           #FB_STATE_MONITOR:
               REGION MONITOR
                   IF #DATA.CMD_MON = 1 THEN
                       IF ("CycleInterrupt_Flag" = TRUE)
                       THEN
                           "CycleInterrupt_Flag" := FALSE;
                           #done := FALSE;
                           #statCMDStateDone := #FB_STATE_MONITOR;
                           FILL_BLK(IN := 16#00,
                                    COUNT := 20,
                                    OUT => #statSendData[0]);

                           #statSendData[0] := 16#02;
                           #statSendData[1] := 'M';
                           #statSendData[2] := 'O';
                           #statSendData[3] := 'N';
                           #statSendData[4] := 16#0D;

                           #statSendTxLength := 5;

                           #statSendReq := TRUE;
                       END_IF;
                   ELSE
                       #statCMDCount := 0;
                       #statCMDState := #statCMDState + 1;
                   END_IF;
               END_REGION MONITOR

           #FB_STATE_FAULT_CLEAR:
               REGION FAULT_CLEAR
                   IF #DATA.CMD_CLR = 1 THEN
                       IF ("CycleInterrupt_Flag" = TRUE)
                       THEN
                           "CycleInterrupt_Flag" := FALSE;
                           #done := FALSE;
                           #statCMDStateDone := #FB_STATE_FAULT_CLEAR;
                           FILL_BLK(IN := 16#00,
                                    COUNT := 20,
                                    OUT => #statSendData[0]);

                           #statSendData[0] := 16#02;
                           #statSendData[1] := 'C';
                           #statSendData[2] := 'L';
                           #statSendData[3] := 'R';
                           #statSendData[4] := 16#0D;

                           #statSendTxLength := 5;

                           #statSendReq := TRUE;
                       END_IF;
                       ELSE
                           #statCMDCount := 0;
                           #statCMDState := #statCMDState + 1;
                       END_IF;

               END_REGION FAULT_CLEAR

           #FB_STATE_REPORT_FAULT:
               REGION REPORT_FAULT
                   IF #DATA.CMD_FLT = 1 THEN
                       IF ("CycleInterrupt_Flag" = TRUE)
                       THEN
                           "CycleInterrupt_Flag" := FALSE;
                           #done := FALSE;
                           #statCMDStateDone := #FB_STATE_REPORT_FAULT;
                           FILL_BLK(IN := 16#00,
                                    COUNT := 20,
                                    OUT => #statSendData[0]);

                           #statSendData[0] := 16#02;
                           #statSendData[1] := 'F';
                           #statSendData[2] := 'L';
                           #statSendData[3] := 'T';
                           #statSendData[4] := 16#0D;

                           #statSendTxLength := 5;

                           #statSendReq := TRUE;
                       END_IF;
                   ELSE
                       #statCMDCount := 0;
                       #statCMDState := #statCMDState + 1;
                   END_IF;
               END_REGION REPORT_FAULT

           #FB_STATE_HV_STATUS:
               REGION HV_STATUS
                   IF #DATA.CMD_STAT = 1 THEN
                       IF ("CycleInterrupt_Flag" = TRUE)
                       THEN
                           "CycleInterrupt_Flag" := FALSE;
                           #done := FALSE;
                           #statCMDStateDone := #FB_STATE_HV_STATUS;
                           FILL_BLK(IN := 16#00,
                                    COUNT := 20,
                                    OUT => #statSendData[0]);

                           #statSendData[0] := 16#02;
                           #statSendData[1] := 'S';
                           #statSendData[2] := 'T';
                           #statSendData[3] := 'A';
                           #statSendData[4] := 'T';

                           #statSendData[5] := 16#0D;

                           #statSendTxLength := 6;

                           #statSendReq := TRUE;
                       END_IF;
                       ELSE
                           #statCMDCount := 0;
                           #statCMDState := #statCMDState + 1;
                       END_IF;
               END_REGION HV_STATUS

           #FB_STATE_X_RAY_ENABLE:
               REGION X_RAY_ENABLE
                   IF #DATA.CMD_ENBL = 1 THEN
                       IF ("CycleInterrupt_Flag" = TRUE)
                       THEN
                           "CycleInterrupt_Flag" := FALSE;
                           #done := FALSE;
                           #statCMDStateDone := #FB_STATE_WD_ENABLE;
                           FILL_BLK(IN := 16#00,
                                    COUNT := 20,
                                    OUT => #statSendData[0]);

                           #statSendData[0] := 16#02;
                           #statSendData[1] := 'E';
                           #statSendData[2] := 'N';
                           #statSendData[3] := 'B';
                           #statSendData[4] := 'L';

                           IF (#DATA.X_RAY_Enable = TRUE) THEN
                               #statSendData[5] := '1';
                           ELSE
                               #statSendData[5] := '0';
                           END_IF;
                           #statSendData[6] := 16#0D;
                           #statSendTxLength := 7;

                           #statSendReq := TRUE;
                       END_IF;
                   ELSE
                       #statCMDCount := 0;
                       #statCMDState := #statCMDState + 1;
                   END_IF;
               END_REGION X_RAY_ENABLE

           #FB_STATE_WD_TIMER:
               REGION WD_TIMER
                   IF #DATA.CMD_WDTE = 1 THEN
                       IF ("CycleInterrupt_Flag" = TRUE)
                       THEN
                           "CycleInterrupt_Flag" := FALSE;
                           #done := FALSE;
                           #statCMDStateDone := #FB_STATE_WD_TIMER;
                           FILL_BLK(IN := 16#00,
                                    COUNT := 20,
                                    OUT => #statSendData[0]);

                           #statSendData[0] := 16#02;
                           #statSendData[1] := 'W';
                           #statSendData[2] := 'D';
                           #statSendData[3] := 'T';
                           #statSendData[4] := 'E';
                           #statSendData[5] := 16#0D;
                           #statSendTxLength := 6;

                           #statSendReq := TRUE;
                       END_IF;
                   ELSE
                       #statCMDCount := 0;
                       #statCMDState := #statCMDState + 1;
                   END_IF;
               END_REGION WD_TIMER            

           #FB_STATE_COMM_PORT_ECHO:
               REGION PORT_ECHO
                   IF #DATA.CMD_FREV = 1 THEN
                       IF ("CycleInterrupt_Flag" = TRUE)
                       THEN
                           "CycleInterrupt_Flag" := FALSE;
                           #done := FALSE;
                           #statCMDStateDone := #FB_STATE_COMM_PORT_ECHO;
                              FILL_BLK(IN := 16#00,
                                       COUNT := 20,
                                       OUT => #statSendData[0]);

                           #statSendData[0] := 16#02;
                           #statSendData[1] := 'F';
                           #statSendData[2] := 'R';
                           #statSendData[3] := 'E';
                           #statSendData[4] := 'V';
                           #statSendData[5] := 16#0D;

                           #statSendTxLength := 6;
                           #statSendReq := TRUE;
                       END_IF;
                   ELSE
                       #statCMDCount := 0;
                       #statCMDState := #statCMDState + 1;
                   END_IF;
               END_REGION PORT_ECHO 

           #FB_STATE_WD_ENABLE:
               REGION WD_ENABLE
                   IF #DATA.CMD_WDOG = 1 THEN
                       IF ("CycleInterrupt_Flag" = TRUE)
                       THEN
                           "CycleInterrupt_Flag" := FALSE;
                           #done := FALSE;
                           #statCMDStateDone := #FB_STATE_WD_ENABLE;
                           FILL_BLK(IN := 16#00,
                                    COUNT := 20,
                                    OUT => #statSendData[0]);

                           #statSendData[0] := 16#02;
                           #statSendData[1] := 'W';
                           #statSendData[2] := 'D';
                           #statSendData[3] := 'O';
                           #statSendData[4] := 'G';

                           IF (#DATA.WDOG = TRUE) THEN
                               #statSendData[5] := '1';
                           ELSE
                               #statSendData[5] := '0';
                           END_IF;
                           #statSendData[6] := 16#0D;
                           #statSendTxLength := 7;

                           #statSendReq := TRUE;
                       END_IF;
                   ELSE
                       #statCMDCount := 0;
                       #statCMDState := #statCMDState + 1;
                   END_IF;
               END_REGION WD_ENABLE 

           #FB_STATE_WD_STATUS:
               REGION WD_STATUS
                   IF #DATA.CMD_WSTAT = 1 THEN
                       REGION Send WD_STATUS Request
                           IF ("CycleInterrupt_Flag" = TRUE)
                           THEN
                               #done := FALSE;
                               "CycleInterrupt_Flag" := FALSE;
                               #statCMDStateDone := #FB_STATE_WD_STATUS;
                               #done := FALSE;
                               FILL_BLK(IN := 16#00,
                               COUNT := 20,
                               OUT => #statSendData[0]);

                               FILL_BLK(IN := 16#00,
                                   COUNT := 50,
                                   OUT => #statRcvData[0]);
                                  #instReceiveP2P.LENGTH := 0;

                               #statSendData[0] := 16#02;
                               #statSendData[1] := 'W';
                               #statSendData[2] := 'S';
                               #statSendData[3] := 'T';
                               #statSendData[4] := 'A';
                               #statSendData[5] := 'T';

                               #statSendData[6] := 16#0D;

                               #statSendTxLength := 7;

                               #statSendReq := TRUE;
                           END_IF;
                       END_REGION Send WD_STATUS Request     
                   ELSE
                       #statCMDCount := 0;
                       #statCMDState := #FB_STATE_VOLTAGE_PROGRAMM;
                   END_IF;
               END_REGION WD_STATUS

           ELSE
               #statCMDState := #FB_STATE_VOLTAGE_PROGRAMM;

       END_CASE;


       IF #debug THEN
           // Statement section IF
           #statCMDCount := 0;
       END_IF;

    END_REGION STATE_MACHINE 

   REGION CALL COMMUNICATION INSTRUCTIONS

       "Send_P2P_DB"(REQ := #statSendReq,
                     "PORT" := #port,
                     BUFFER := #statSendData,
                     LENGTH := #statSendTxLength,
                     DONE => #statRS232TxDone,
                     ERROR => #statRS232Error,
                     STATUS => #statRS232Status);

       "Receive_P2P_DB"("PORT" := #port,
                        BUFFER := #statRcvData,
                        NDR => #statRS232Ndr,
                        ERROR => #statRS232Error,
                        STATUS => #statRS232Status,
                        LENGTH => #statSendRxLength);


   END_REGION CALL COMMUNICATION INSTRUCTIONS

   //Reset request has been sent
   IF #statRS232TxDone
   THEN
       #statSendReq := false;
   END_IF;

   IF #statRS232Ndr
   THEN
       #statStatus:= #statRS232Status;

       #statCMDCount := #statCMDCount + 1;

       IF (#statRS232Status = #STATUS_msg_timeout) OR (#statRS232Status = "STATUS_msg_CHAR_timeout") THEN
           CASE #statCMDState OF

               #FB_STATE_VOLTAGE_PROGRAMM:
                   REGION Recive Voltage Programm

                       IF #statSendRxLength = 8
                           AND #statRcvData[0] = #statSendData[0]
                           AND #statRcvData[1] = #statSendData[1]
                           AND #statRcvData[2] = #statSendData[2]
                           AND #statRcvData[3] = #statSendData[3]
                           AND #statRcvData[4] = #statSendData[4]
                           AND #statRcvData[5] = #statSendData[5]
                           AND #statRcvData[6] = #statSendData[6]
                           AND #statRcvData[7] = #statSendData[7]
                       THEN
                           #statCMDState := #statCMDState + 1;

                     //      IF NOT #DATA.CMD_CYCLE THEN
                           #DATA.CMD_VP := FALSE;
                           #DATA.CMD_VP_Ok := TRUE;
                      //     END_IF;
                       END_IF;
                   END_REGION Recive Voltage Programm       

               #FB_STATE_CURRENT_PROGRAMM:
                   REGION Recive Current Programm Request

                       IF #statSendRxLength = 8
                           AND #statRcvData[0] = #statSendData[0]
                           AND #statRcvData[1] = #statSendData[1]
                           AND #statRcvData[2] = #statSendData[2]
                           AND #statRcvData[3] = #statSendData[3]
                           AND #statRcvData[4] = #statSendData[4]
                           AND #statRcvData[5] = #statSendData[5]
                           AND #statRcvData[6] = #statSendData[6]
                       THEN
                           #statCMDState := #statCMDState + 1;
                   //        IF NOT #DATA.CMD_CYCLE THEN
                           #DATA.CMD_CP := FALSE;
                           #DATA.CMD_CP_Ok := TRUE;
                    //       END_IF;
                       END_IF;
                   END_REGION Recive Current Programm Request           

               #FB_STATE_MONITOR:
                   REGION Recive MONITOR Request
                       IF NOT #DATA.CMD_CYCLE THEN
                           #DATA.CMD_MON := FALSE;
                       END_IF;
                       IF #statSendRxLength = 21
                       THEN
                           //Вставить код для обработки ответа
                           //Преобразование V monitor
                           Chars_TO_Strg(Chars := #statRcvData,
          pChars := 1,
          Cnt := 4,
          Strg => #statString);
                           STRG_VAL(IN := #statString,
          FORMAT := 0,
          P := 1,
          OUT => #temp_Uint);
   #DATA.VP_Monitor := UINT_TO_REAL(#temp_Uint);
                           #DATA.VP_Monitor := #DATA.VP_Monitor / 10.0;

                           //Преобразование I monitor
                           Chars_TO_Strg(Chars := #statRcvData,
          pChars := 6,
          Cnt := 5,
          Strg => #statString);
                           STRG_VAL(IN := #statString,
          FORMAT := 0,
          P := 1,
          OUT => #temp_Uint);
                               #DATA.CP_Monitor := #temp_Uint;


                           //Преобразование T monitor
                           Chars_TO_Strg(Chars := #statRcvData,
          pChars := 12,
          Cnt := 4,
          Strg => #statString);
                           STRG_VAL(IN := #statString,
          FORMAT := 0,
          P := 1,
          OUT => #temp_Uint);
                           #DATA.T_Monitor := UINT_TO_REAL(#temp_Uint);
                           #DATA.T_Monitor := #DATA.T_Monitor / 10.0;

                           //Преобразование Filament monitor
                           Chars_TO_Strg(Chars := #statRcvData,
          pChars := 17,
          Cnt := 4,
          Strg => #statString);
                           STRG_VAL(IN := #statString,
          FORMAT := 0,
          P := 1,
          OUT => #temp_Uint);
                           #DATA.FIL_Monitor := #temp_Uint;

                           #statCMDState := #statCMDState + 1;
                       END_IF;
                   END_REGION Recive MONITOR Request 

               #FB_STATE_FAULT_CLEAR:
                   REGION Recive FAULT_CLEAR Request
                       IF NOT #DATA.CMD_CYCLE THEN
                           #DATA.CMD_CLR := FALSE;
                       END_IF;
                       IF #statRcvData[0] = #statSendData[0]
                           AND #statRcvData[1] = #statSendData[1]
                           AND #statRcvData[2] = #statSendData[2]
                           AND #statRcvData[3] = #statSendData[3]
                           AND #statRcvData[4] = #statSendData[4]
                       THEN
                           #statCMDCount := 0;
                           #statCMDState := #statCMDState + 1;
                       END_IF;
                   END_REGION Recive FAULT_CLEAR Request   

               #FB_STATE_REPORT_FAULT:
                   REGION Recive REPORT_FAULT Request
                       IF NOT #DATA.CMD_CYCLE THEN
                           #DATA.CMD_FLT := FALSE;
                       END_IF;
                       IF #statSendRxLength = 19
                       THEN
                           //Вставить код для обработки ответа
                           IF #statRcvData[1] = '1' THEN
                               #DATA.FLT[0] := TRUE;
                           ELSE
                               #DATA.FLT[0] := FALSE;
                           END_IF;

                           IF #statRcvData[3] = '1' THEN
                               #DATA.FLT[1] := TRUE;
                           ELSE
                               #DATA.FLT[1] := FALSE;
                           END_IF;

                           IF #statRcvData[5] = '1' THEN
                               #DATA.FLT[2] := TRUE;
                           ELSE
                               #DATA.FLT[2] := FALSE;
                           END_IF;

                           IF #statRcvData[7] = '1' THEN
                               #DATA.FLT[3] := TRUE;
                           ELSE
                               #DATA.FLT[3] := FALSE;
                           END_IF;

                           IF #statRcvData[9] = '1' THEN
                               #DATA.FLT[4] := TRUE;
                           ELSE
                               #DATA.FLT[4] := FALSE;
                           END_IF;

                           IF #statRcvData[11] = '1' THEN
                               #DATA.FLT[5] := TRUE;
                           ELSE
                               #DATA.FLT[5] := FALSE;
                           END_IF;

                           IF #statRcvData[13] = '1' THEN
                               #DATA.FLT[6] := TRUE;
                           ELSE
                               #DATA.FLT[6] := FALSE;
                           END_IF;

                           IF #statRcvData[15] = '1' THEN
                               #DATA.FLT[7] := TRUE;
                           ELSE
                               #DATA.FLT[7] := FALSE;
                           END_IF;

                           IF #statRcvData[17] = '1' THEN
                               #DATA.FLT[8] := TRUE;
                           ELSE
                               #DATA.FLT[8] := FALSE;
                           END_IF;

                           #statCMDState := #statCMDState + 1;
                       END_IF;
                   END_REGION Recive REPORT_FAULT Request   

               #FB_STATE_HV_STATUS:
                   REGION Recive MONITOR Reques                
                       IF NOT #DATA.CMD_CYCLE THEN
                           #DATA.CMD_STAT := FALSE;
                       END_IF;
                       IF #statSendRxLength = 3
                       THEN
                           IF (#statRcvData[1] = '1') THEN
                               #DATA.X_RAY_Status := TRUE;
                           ELSE
                               #DATA.X_RAY_Status := FALSE;
                           END_IF;
                           #statCMDCount := 0;
                           #statCMDState := #statCMDState + 1;
                       END_IF;
                   END_REGION Recive HV_STATUS Request  

               #FB_STATE_X_RAY_ENABLE:
                   REGION Recive X_RAY_ENABLE Request
                       IF NOT #DATA.CMD_CYCLE THEN
                           #DATA.CMD_ENBL := FALSE;
                       END_IF;
                       IF  (#statSendRxLength = 7)
                           AND #statRcvData[1] = #statSendData[1]
                           AND #statRcvData[2] = #statSendData[2]
                           AND #statRcvData[3] = #statSendData[3]
                           AND #statRcvData[4] = #statSendData[4]
                       THEN
                           IF #statRcvData[5] = '1' THEN
                               #DATA.X_RAY_Enable := TRUE;
                           ELSE
                               #DATA.X_RAY_Enable := FALSE;
                           END_IF;
                           #statCMDCount := 0;
                           #statCMDState := #statCMDState + 1;
                       END_IF;
                   END_REGION Recive X_RAY_ENABLE Request 

               #FB_STATE_WD_TIMER:
                   REGION Recive WD_TIMER Request
                       IF NOT #DATA.CMD_CYCLE THEN
                           #DATA.CMD_WDTE := FALSE;
                       END_IF;
                       IF (#statSendRxLength = 4)
                           AND #statRcvData[1] = 'O'
                           AND #statRcvData[2] = 'K'
                       THEN
                           #DATA.WDTE := TRUE;
                           #statCMDCount := 0;
                           #statCMDState := #statCMDState + 1;
                       END_IF;
                   END_REGION Recive WD_TIMER Request 

               #FB_STATE_COMM_PORT_ECHO:
                   REGION Recive PORT_ECHO Request
                       IF NOT #DATA.CMD_CYCLE THEN
                           #DATA.CMD_FREV := FALSE;
                       END_IF;
                       IF #statSendRxLength = 6
                           AND #statRcvData[1] = 16#32
                           AND #statRcvData[2] = 16#30
                           AND #statRcvData[3] = 16#30
                           AND #statRcvData[4] = 16#30
                       THEN
                           //Вставить код для обработки ответа
                           #DATA.FREV := TRUE;
                           #statCMDCount := 0;
                           #statCMDState := #statCMDState + 1;
                       END_IF;
                   END_REGION Recive PORT_ECHO Request  

               #FB_STATE_WD_ENABLE:
                   REGION Recive WD_ENABLE Request
                       IF NOT #DATA.CMD_CYCLE THEN
                           #DATA.CMD_WDOG := FALSE;
                       END_IF;
                       IF #statSendRxLength = 7
                           AND #statRcvData[0] = #statSendData[0]
                           AND #statRcvData[1] = #statSendData[1]
                           AND #statRcvData[2] = #statSendData[2]
                           AND #statRcvData[3] = #statSendData[3]
                           AND #statRcvData[4] = #statSendData[4]
                       THEN
                           IF #statRcvData[5] = '1' THEN
                               #DATA.WDOG := TRUE;
                           ELSE
                               #DATA.WDOG := FALSE;
                           END_IF;
                           #statCMDCount := 0;
                           #statCMDState := #statCMDState + 1;
                       END_IF;
                       END_REGION Recive WD_ENABLE Request  

               #FB_STATE_WD_STATUS:
                   REGION Recive WD_STATUS    
                       IF #statSendRxLength = 3
                       THEN
                           IF NOT #DATA.CMD_CYCLE THEN
                               #DATA.CMD_WSTAT := FALSE;
                           END_IF;
                           IF (#statRcvData[1] = '1') THEN
                               #DATA.WDOG_Status := TRUE;
                           ELSE
                               #DATA.WDOG_Status := FALSE;
                           END_IF;
                           #statCMDState := #FB_STATE_VOLTAGE_PROGRAMM;
                       END_IF;
                   END_REGION Recive WD_STATUS
               ELSE
                   REGION undefined state        
                       #statCMDState := #FB_STATE_VOLTAGE_PROGRAMM;
                   END_REGION undefined state    
           END_CASE;
           #statCMDCount := 0;
           #statError := FALSE;
       ELSE
           #statError := TRUE;
           #statCMDCount := #statCMDCount +1;
           IF #statCMDCount >= "CountERR" THEN
               #statCMDState := #FB_STATE_NO_PROCESSING;
               #DATA.DiagnosticCMD[#statCMDState].status := #statStatus;
               #DATA.DiagnosticCMD[#statCMDState].count := #statCMDCount;
           END_IF;
       END_IF;
   END_IF;

   REGION OUTPUT  
       REGION Write static values to outputs

           #error := #statError;
           #status := #statStatus;
           IF (NOT #error)
               AND ((#statRS232TxDone AND #debug) OR (#statRS232Ndr AND (#statStatus <> #ERR_Response_Generator)))
           THEN
               #done := TRUE;
           END_IF;

           #DATA.DiagnosticCMD[#statCMDState].status := #status;
           #DATA.DiagnosticCMD[#statCMDState].count := #statCMDCount + 1;

           #done_CMD := #statCMDState;

           ENO := TRUE;

       END_REGION Write static values to outputs
   END_REGION OUTPUTS
END_FUNCTION_BLOCK

FUNCTION_BLOCK "GenOperate"   // FB8, LAD
{ S7_Optimized_Access := 'TRUE' }
VERSION : 0.1
   VAR_INPUT
      cmdXRAY : Bool;
      interLock : Bool;
      statusGEN : Bool;
      resset : Bool;
      HW_PORT : Port;
      SelGen1 : Bool;
      SelGen2 : Bool;
   END_VAR
   VAR_OUTPUT
      "X-RAY_HL" : Bool;
      POWER_Status : Bool;
      Fault : Bool;
      Ready : Bool;
      Status : Word;
   END_VAR
   VAR_IN_OUT
      DATA_Generator : "typeGeneratorDATA";
   END_VAR
   VAR
      err_CMD_Generator : Bool;
      status_CMD_Gnerator : UInt;
      err_Check_Presset : Bool;
      done_CMD_Generator : Bool;
      status_POWER_OK : Bool;
      status_Delta_VP : Real;
      status_Delta_CP : Real;
      reset_Generator : Bool;
      noACK : Bool;
      Front1 : Bool;
      Front2 : Bool;
      Rise1 : Bool;
   END_VAR
   VAR_TEMP   // added for the SCL form of the ladder/FBD networks
      _w1 : Bool;
      _w2 : Bool;
      _w3 : Bool;
   END_VAR
BEGIN

REGION Network 1: Command HV Status
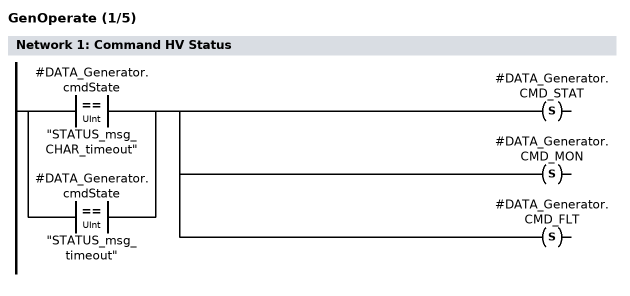
   RUNG wire#powerrail
      { S7_Templates := "SrcType := UInt" } EQ_Contact(in1 := #DATA_Generator.cmdState, in2 := "STATUS_msg_CHAR_timeout")
      wire#w1
      S_Coil( #DATA_Generator.CMD_STAT )
   END_RUNG
   RUNG wire#powerrail
      { S7_Templates := "SrcType := UInt" } EQ_Contact(in1 := #DATA_Generator.cmdState, in2 := "STATUS_msg_timeout")
   END_RUNG wire#w1
   RUNG wire#w1
      S_Coil( #DATA_Generator.CMD_MON )
   END_RUNG
   RUNG wire#w1
      S_Coil( #DATA_Generator.CMD_FLT )
   END_RUNG
   // the same network as SCL:
   IF (#DATA_Generator.cmdState = "STATUS_msg_CHAR_timeout") OR (#DATA_Generator.cmdState = "STATUS_msg_timeout") THEN
       #DATA_Generator.CMD_STAT := TRUE;
       #DATA_Generator.CMD_MON := TRUE;
       #DATA_Generator.CMD_FLT := TRUE;
   END_IF;
END_REGION

REGION Network 2: Когда нет ответа от генератора, то сбрасываем блок работы с генератором
   // Проверка соединения с генератором. Если при выполнении команды получаем ошибку по таймауту ответа от генератора, то сбрасываем интерфейс обмена с генератором, включаем режим DEBUG (при отутствии ответа от генератора не останавливаем обмен), цстанавливаем циклический обмен и запускаем команду на получения ECHO. Как только по команде получения ECHO мы получаем ответ от генератора, то сбрасываем команду на получения ECHO, а выставляем команду Monitor и WD. Получаем фактическое значение напряжения и тока генератора, читаем сторожевой таймер
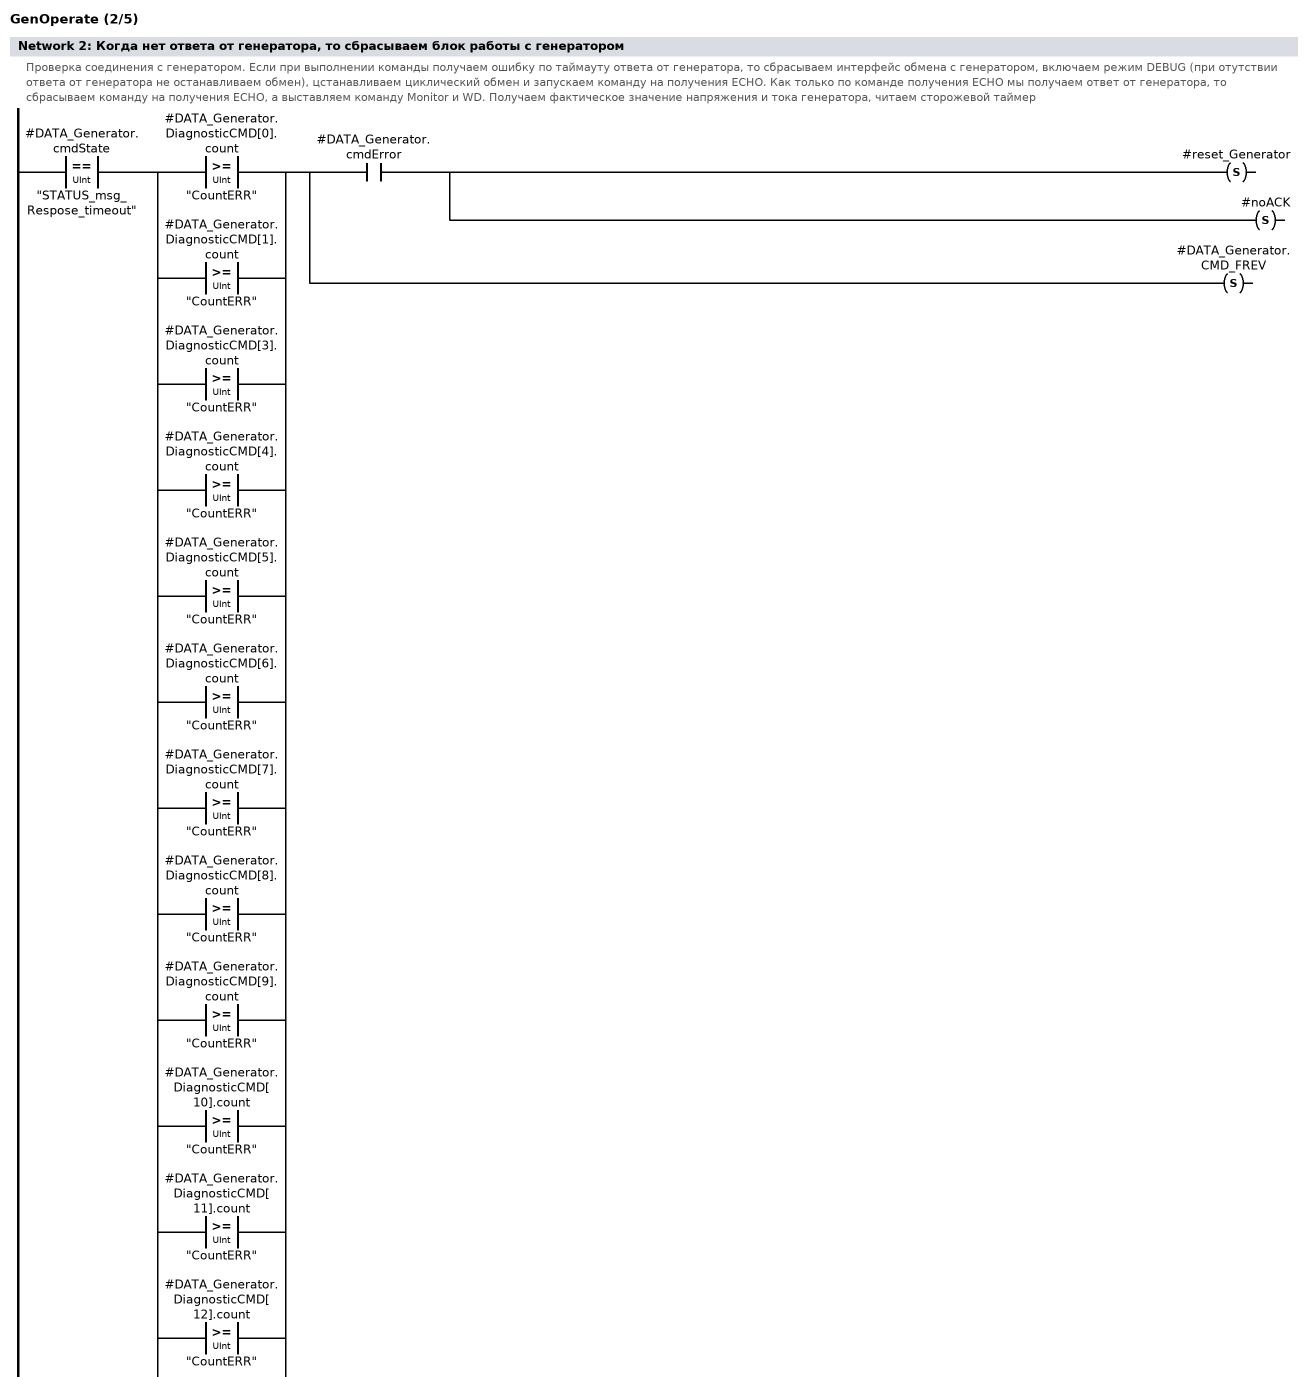
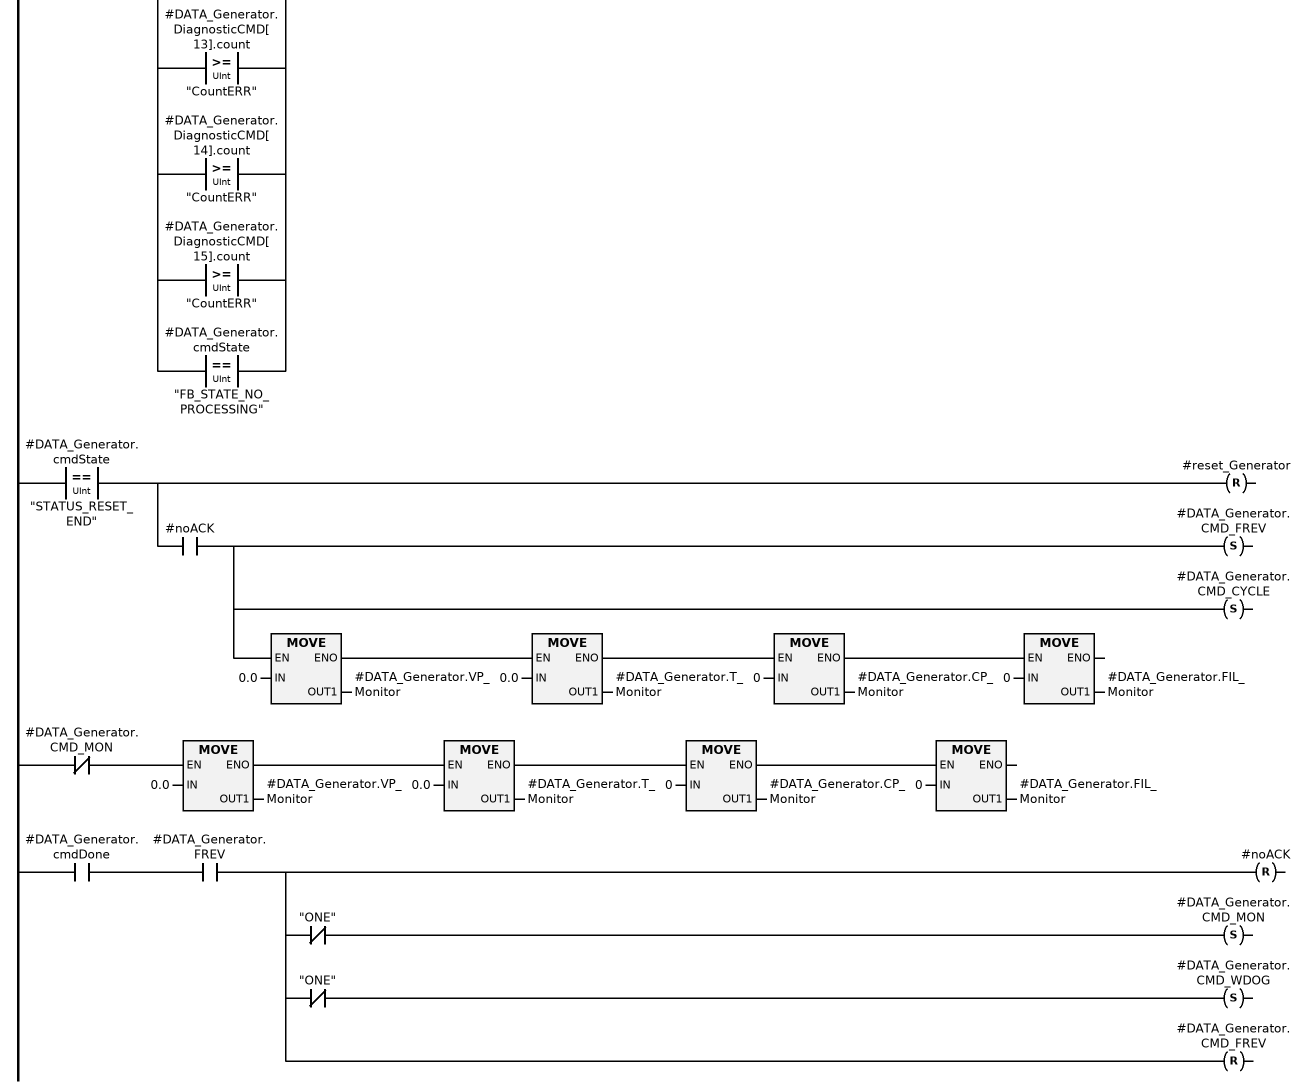
   RUNG wire#powerrail
      { S7_Templates := "SrcType := UInt" } EQ_Contact(in1 := #DATA_Generator.cmdState, in2 := "STATUS_msg_Respose_timeout")
      wire#w1
      { S7_Templates := "SrcType := UInt" } GE_Contact(in1 := #DATA_Generator.DiagnosticCMD[0].count, in2 := "CountERR")
      wire#w2
      Contact( #DATA_Generator.cmdError )
      wire#w3
      S_Coil( #reset_Generator )
   END_RUNG
   RUNG wire#w1
      { S7_Templates := "SrcType := UInt" } GE_Contact(in1 := #DATA_Generator.DiagnosticCMD[1].count, in2 := "CountERR")
   END_RUNG wire#w2
   RUNG wire#w1
      { S7_Templates := "SrcType := UInt" } GE_Contact(in1 := #DATA_Generator.DiagnosticCMD[3].count, in2 := "CountERR")
   END_RUNG wire#w2
   RUNG wire#w1
      { S7_Templates := "SrcType := UInt" } GE_Contact(in1 := #DATA_Generator.DiagnosticCMD[4].count, in2 := "CountERR")
   END_RUNG wire#w2
   RUNG wire#w1
      { S7_Templates := "SrcType := UInt" } GE_Contact(in1 := #DATA_Generator.DiagnosticCMD[5].count, in2 := "CountERR")
   END_RUNG wire#w2
   RUNG wire#w1
      { S7_Templates := "SrcType := UInt" } GE_Contact(in1 := #DATA_Generator.DiagnosticCMD[6].count, in2 := "CountERR")
   END_RUNG wire#w2
   RUNG wire#w1
      { S7_Templates := "SrcType := UInt" } GE_Contact(in1 := #DATA_Generator.DiagnosticCMD[7].count, in2 := "CountERR")
   END_RUNG wire#w2
   RUNG wire#w1
      { S7_Templates := "SrcType := UInt" } GE_Contact(in1 := #DATA_Generator.DiagnosticCMD[8].count, in2 := "CountERR")
   END_RUNG wire#w2
   RUNG wire#w1
      { S7_Templates := "SrcType := UInt" } GE_Contact(in1 := #DATA_Generator.DiagnosticCMD[9].count, in2 := "CountERR")
   END_RUNG wire#w2
   RUNG wire#w1
      { S7_Templates := "SrcType := UInt" } GE_Contact(in1 := #DATA_Generator.DiagnosticCMD[10].count, in2 := "CountERR")
   END_RUNG wire#w2
   RUNG wire#w1
      { S7_Templates := "SrcType := UInt" } GE_Contact(in1 := #DATA_Generator.DiagnosticCMD[11].count, in2 := "CountERR")
   END_RUNG wire#w2
   RUNG wire#w1
      { S7_Templates := "SrcType := UInt" } GE_Contact(in1 := #DATA_Generator.DiagnosticCMD[12].count, in2 := "CountERR")
   END_RUNG wire#w2
   RUNG wire#w1
      { S7_Templates := "SrcType := UInt" } GE_Contact(in1 := #DATA_Generator.DiagnosticCMD[13].count, in2 := "CountERR")
   END_RUNG wire#w2
   RUNG wire#w1
      { S7_Templates := "SrcType := UInt" } GE_Contact(in1 := #DATA_Generator.DiagnosticCMD[14].count, in2 := "CountERR")
   END_RUNG wire#w2
   RUNG wire#w1
      { S7_Templates := "SrcType := UInt" } GE_Contact(in1 := #DATA_Generator.DiagnosticCMD[15].count, in2 := "CountERR")
   END_RUNG wire#w2
   RUNG wire#w1
      { S7_Templates := "SrcType := UInt" } EQ_Contact(in1 := #DATA_Generator.cmdState, in2 := "FB_STATE_NO_PROCESSING")
   END_RUNG wire#w2
   RUNG wire#w3
      S_Coil( #noACK )
   END_RUNG
   RUNG wire#w2
      S_Coil( #DATA_Generator.CMD_FREV )
   END_RUNG
   RUNG wire#powerrail
      { S7_Templates := "SrcType := UInt" } EQ_Contact(in1 := #DATA_Generator.cmdState, in2 := "STATUS_RESET_END")
      wire#w4
      R_Coil( #reset_Generator )
   END_RUNG
   RUNG wire#w4
      Contact( #noACK )
      wire#w5
      S_Coil( #DATA_Generator.CMD_FREV )
   END_RUNG
   RUNG wire#w5
      S_Coil( #DATA_Generator.CMD_CYCLE )
   END_RUNG
   RUNG wire#w5
      Move(in := 0.0, out1 => #DATA_Generator.VP_Monitor)
      Move(in := 0.0, out1 => #DATA_Generator.T_Monitor)
      Move(in := 0, out1 => #DATA_Generator.CP_Monitor)
      Move(in := 0, out1 => #DATA_Generator.FIL_Monitor)
   END_RUNG
   RUNG wire#powerrail
      I_Contact( #DATA_Generator.CMD_MON )
      Move(in := 0.0, out1 => #DATA_Generator.VP_Monitor)
      Move(in := 0.0, out1 => #DATA_Generator.T_Monitor)
      Move(in := 0, out1 => #DATA_Generator.CP_Monitor)
      Move(in := 0, out1 => #DATA_Generator.FIL_Monitor)
   END_RUNG
   RUNG wire#powerrail
      Contact( #DATA_Generator.cmdDone )
      Contact( #DATA_Generator.FREV )
      wire#w6
      R_Coil( #noACK )
   END_RUNG
   RUNG wire#w6
      I_Contact( "ONE" )
      S_Coil( #DATA_Generator.CMD_MON )
   END_RUNG
   RUNG wire#w6
      I_Contact( "ONE" )
      S_Coil( #DATA_Generator.CMD_WDOG )
   END_RUNG
   RUNG wire#w6
      R_Coil( #DATA_Generator.CMD_FREV )
   END_RUNG
   // the same network as SCL:
   #_w1 := (#DATA_Generator.cmdState = "STATUS_msg_Respose_timeout") AND ((#DATA_Generator.DiagnosticCMD[0].count >= "CountERR") OR (#DATA_Generator.DiagnosticCMD[1].count >= "CountERR") OR (#DATA_Generator.DiagnosticCMD[3].count >= "CountERR") OR (#DATA_Generator.DiagnosticCMD[4].count >= "CountERR") OR (#DATA_Generator.DiagnosticCMD[5].count >= "CountERR") OR (#DATA_Generator.DiagnosticCMD[6].count >= "CountERR") OR (#DATA_Generator.DiagnosticCMD[7].count >= "CountERR") OR (#DATA_Generator.DiagnosticCMD[8].count >= "CountERR") OR (#DATA_Generator.DiagnosticCMD[9].count >= "CountERR") OR (#DATA_Generator.DiagnosticCMD[10].count >= "CountERR") OR (#DATA_Generator.DiagnosticCMD[11].count >= "CountERR") OR (#DATA_Generator.DiagnosticCMD[12].count >= "CountERR") OR (#DATA_Generator.DiagnosticCMD[13].count >= "CountERR") OR (#DATA_Generator.DiagnosticCMD[14].count >= "CountERR") OR (#DATA_Generator.DiagnosticCMD[15].count >= "CountERR") OR (#DATA_Generator.cmdState = "FB_STATE_NO_PROCESSING"));
   IF #_w1 AND #DATA_Generator.cmdError THEN
       #reset_Generator := TRUE;
       #noACK := TRUE;
   END_IF;
   IF #_w1 THEN #DATA_Generator.CMD_FREV := TRUE; END_IF;
   #_w2 := #DATA_Generator.cmdState = "STATUS_RESET_END";
   IF #_w2 THEN #reset_Generator := FALSE; END_IF;
   IF #_w2 AND #noACK THEN
       #DATA_Generator.CMD_FREV := TRUE;
       #DATA_Generator.CMD_CYCLE := TRUE;
       #DATA_Generator.VP_Monitor := 0.0;
       #DATA_Generator.T_Monitor := 0.0;
       #DATA_Generator.CP_Monitor := 0;
       #DATA_Generator.FIL_Monitor := 0;
   END_IF;
   IF NOT #DATA_Generator.CMD_MON THEN
       #DATA_Generator.VP_Monitor := 0.0;
       #DATA_Generator.T_Monitor := 0.0;
       #DATA_Generator.CP_Monitor := 0;
       #DATA_Generator.FIL_Monitor := 0;
   END_IF;
   #_w3 := #DATA_Generator.cmdDone AND #DATA_Generator.FREV;
   IF #_w3 THEN #noACK := FALSE; END_IF;
   IF #_w3 AND NOT "ONE" THEN
       #DATA_Generator.CMD_MON := TRUE;
       #DATA_Generator.CMD_WDOG := TRUE;
   END_IF;
   IF #_w3 THEN #DATA_Generator.CMD_FREV := FALSE; END_IF;
END_REGION

REGION Network 3: Включение X-RAY
   // По сигналу устанавливаем:
   // 1. Команду программирования Напряжения и Тока в генераторе
   // 2. Сброс статуса выполнения команды на программирование Напряджения и Тока
   // 3. После выполнения команды программирования Напряжения и Тока выставляем статус выполнения команд
   // 4. Пос статусу выполнения команды устанавливаем команду на включение генаратора
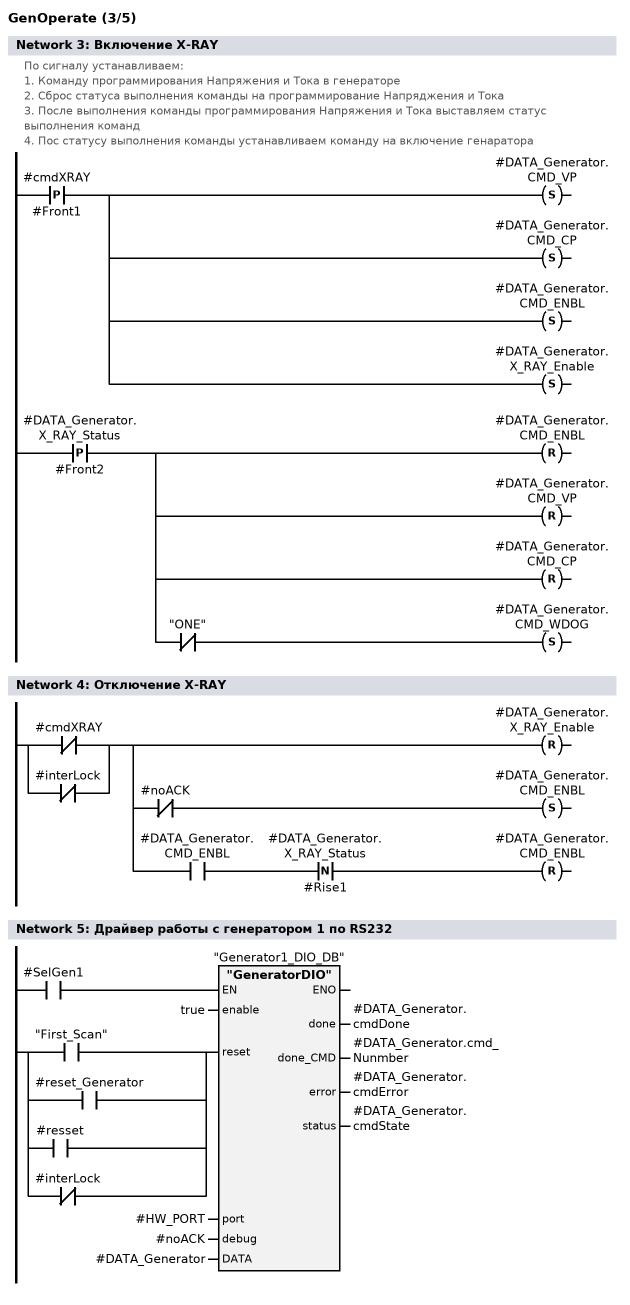
   RUNG wire#powerrail
      P_Contact(operand := #cmdXRAY, bit := #Front1)
      wire#w1
      S_Coil( #DATA_Generator.CMD_VP )
   END_RUNG
   RUNG wire#w1
      S_Coil( #DATA_Generator.CMD_CP )
   END_RUNG
   RUNG wire#w1
      S_Coil( #DATA_Generator.CMD_ENBL )
   END_RUNG
   RUNG wire#w1
      S_Coil( #DATA_Generator.X_RAY_Enable )
   END_RUNG
   RUNG wire#powerrail
      P_Contact(operand := #DATA_Generator.X_RAY_Status, bit := #Front2)
      wire#w2
      R_Coil( #DATA_Generator.CMD_ENBL )
   END_RUNG
   RUNG wire#w2
      R_Coil( #DATA_Generator.CMD_VP )
   END_RUNG
   RUNG wire#w2
      R_Coil( #DATA_Generator.CMD_CP )
   END_RUNG
   RUNG wire#w2
      I_Contact( "ONE" )
      S_Coil( #DATA_Generator.CMD_WDOG )
   END_RUNG
   // the same network as SCL:
   #_w1 := #cmdXRAY AND NOT #Front1;   // rising edge of #cmdXRAY
   #Front1 := #cmdXRAY;
   IF #_w1 THEN
       #DATA_Generator.CMD_VP := TRUE;
       #DATA_Generator.CMD_CP := TRUE;
       #DATA_Generator.CMD_ENBL := TRUE;
       #DATA_Generator.X_RAY_Enable := TRUE;
   END_IF;
   #_w2 := #DATA_Generator.X_RAY_Status AND NOT #Front2;   // rising edge of #DATA_Generator.X_RAY_Status
   #Front2 := #DATA_Generator.X_RAY_Status;
   IF #_w2 THEN
       #DATA_Generator.CMD_ENBL := FALSE;
       #DATA_Generator.CMD_VP := FALSE;
       #DATA_Generator.CMD_CP := FALSE;
   END_IF;
   IF #_w2 AND NOT "ONE" THEN #DATA_Generator.CMD_WDOG := TRUE; END_IF;
END_REGION

REGION Network 4: Отключение X-RAY
   RUNG wire#powerrail
      I_Contact( #cmdXRAY )
      wire#w1
      R_Coil( #DATA_Generator.X_RAY_Enable )
   END_RUNG
   RUNG wire#powerrail
      I_Contact( #interLock )
   END_RUNG wire#w1
   RUNG wire#w1
      I_Contact( #noACK )
      S_Coil( #DATA_Generator.CMD_ENBL )
   END_RUNG
   RUNG wire#w1
      Contact( #DATA_Generator.CMD_ENBL )
      N_Contact(operand := #DATA_Generator.X_RAY_Status, bit := #Rise1)
      R_Coil( #DATA_Generator.CMD_ENBL )
   END_RUNG
   // the same network as SCL:
   #_w1 := NOT #cmdXRAY OR NOT #interLock;
   IF #_w1 THEN #DATA_Generator.X_RAY_Enable := FALSE; END_IF;
   IF #_w1 AND NOT #noACK THEN #DATA_Generator.CMD_ENBL := TRUE; END_IF;
   #_w2 := #_w1 AND #DATA_Generator.CMD_ENBL AND NOT #DATA_Generator.X_RAY_Status AND #Rise1;   // falling edge of #DATA_Generator.X_RAY_Status
   #Rise1 := #DATA_Generator.X_RAY_Status;
   IF #_w2 THEN #DATA_Generator.CMD_ENBL := FALSE; END_IF;
END_REGION

REGION Network 5: Драйвер работы с генератором 1 по RS232
   RUNG wire#powerrail
      Contact( #SelGen1 )
      "Generator1_DIO_DB"(reset := wire#w1, enable := true, port := #HW_PORT, debug := #noACK, DATA := #DATA_Generator, done => #DATA_Generator.cmdDone, done_CMD => #DATA_Generator.cmd_Nunmber, error => #DATA_Generator.cmdError, status => #DATA_Generator.cmdState)
   END_RUNG
   RUNG wire#powerrail
      Contact( "First_Scan" )
   END_RUNG wire#w1
   RUNG wire#powerrail
      Contact( #reset_Generator )
   END_RUNG wire#w1
   RUNG wire#powerrail
      Contact( #resset )
   END_RUNG wire#w1
   RUNG wire#powerrail
      I_Contact( #interLock )
   END_RUNG wire#w1
   // the same network as SCL:
   IF #SelGen1 THEN
       "Generator1_DIO_DB"(enable := true,   // "GeneratorDIO"
                           reset := "First_Scan" OR #reset_Generator OR #resset OR NOT #interLock,
                           port := #HW_PORT,
                           debug := #noACK,
                           DATA := #DATA_Generator,
                           done => #DATA_Generator.cmdDone,
                           done_CMD => #DATA_Generator.cmd_Nunmber,
                           error => #DATA_Generator.cmdError,
                           status => #DATA_Generator.cmdState);
   END_IF;
END_REGION

REGION Network 6: Драйвер работы с генератором 2 по RS232
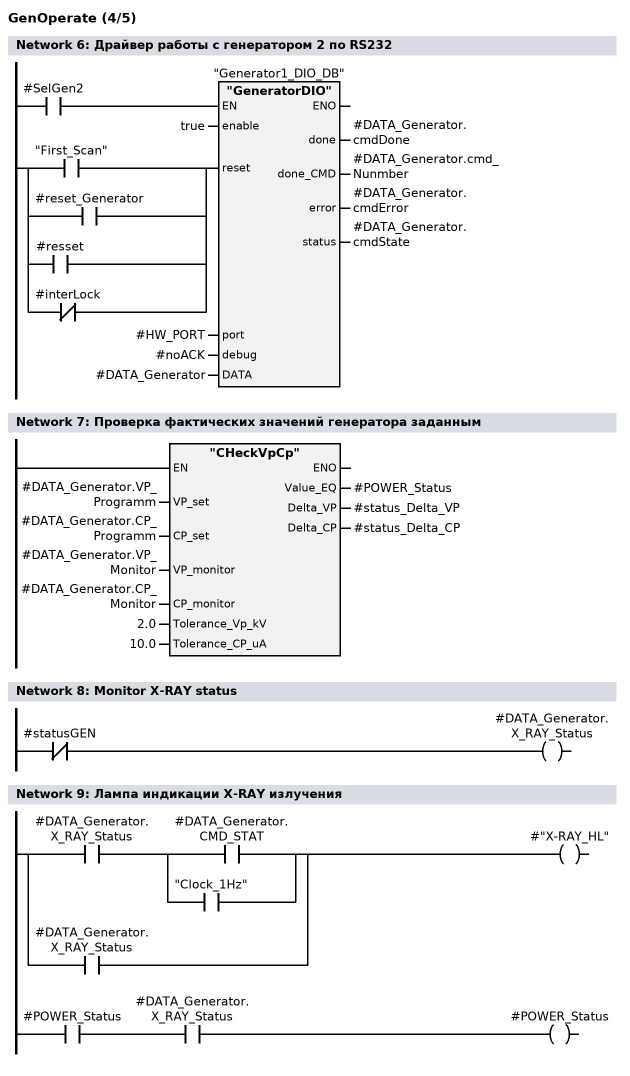
   RUNG wire#powerrail
      Contact( #SelGen2 )
      "Generator1_DIO_DB"(reset := wire#w1, enable := true, port := #HW_PORT, debug := #noACK, DATA := #DATA_Generator, done => #DATA_Generator.cmdDone, done_CMD => #DATA_Generator.cmd_Nunmber, error => #DATA_Generator.cmdError, status => #DATA_Generator.cmdState)
   END_RUNG
   RUNG wire#powerrail
      Contact( "First_Scan" )
   END_RUNG wire#w1
   RUNG wire#powerrail
      Contact( #reset_Generator )
   END_RUNG wire#w1
   RUNG wire#powerrail
      Contact( #resset )
   END_RUNG wire#w1
   RUNG wire#powerrail
      I_Contact( #interLock )
   END_RUNG wire#w1
   // the same network as SCL:
   IF #SelGen2 THEN
       "Generator1_DIO_DB"(enable := true,   // "GeneratorDIO"
                           reset := "First_Scan" OR #reset_Generator OR #resset OR NOT #interLock,
                           port := #HW_PORT,
                           debug := #noACK,
                           DATA := #DATA_Generator,
                           done => #DATA_Generator.cmdDone,
                           done_CMD => #DATA_Generator.cmd_Nunmber,
                           error => #DATA_Generator.cmdError,
                           status => #DATA_Generator.cmdState);
   END_IF;
END_REGION

REGION Network 7: Проверка фактических значений генератора заданным
   RUNG wire#powerrail
      "CHeckVpCp"(VP_set := #DATA_Generator.VP_Programm, CP_set := #DATA_Generator.CP_Programm, VP_monitor := #DATA_Generator.VP_Monitor, CP_monitor := #DATA_Generator.CP_Monitor, Tolerance_Vp_kV := 2.0, Tolerance_CP_uA := 10.0, Value_EQ => #POWER_Status, Delta_VP => #status_Delta_VP, Delta_CP => #status_Delta_CP)
   END_RUNG
   // the same network as SCL:
   "CHeckVpCp"(VP_set := #DATA_Generator.VP_Programm,
               CP_set := #DATA_Generator.CP_Programm,
               VP_monitor := #DATA_Generator.VP_Monitor,
               CP_monitor := #DATA_Generator.CP_Monitor,
               Tolerance_Vp_kV := 2.0,
               Tolerance_CP_uA := 10.0,
               Value_EQ => #POWER_Status,
               Delta_VP => #status_Delta_VP,
               Delta_CP => #status_Delta_CP);
END_REGION

REGION Network 8: Monitor X-RAY status
   RUNG wire#powerrail
      I_Contact( #statusGEN )
      Coil( #DATA_Generator.X_RAY_Status )
   END_RUNG
   // the same network as SCL:
   #DATA_Generator.X_RAY_Status := NOT #statusGEN;
END_REGION

REGION Network 9: Лампа индикации X-RAY излучения
   RUNG wire#powerrail
      Contact( #DATA_Generator.X_RAY_Status )
      wire#w1
      Contact( #DATA_Generator.CMD_STAT )
      wire#w2
      Coil( #"X-RAY_HL" )
   END_RUNG
   RUNG wire#w1
      Contact( "Clock_1Hz" )
   END_RUNG wire#w2
   RUNG wire#powerrail
      Contact( #DATA_Generator.X_RAY_Status )
   END_RUNG wire#w2
   RUNG wire#powerrail
      Contact( #POWER_Status )
      Contact( #DATA_Generator.X_RAY_Status )
      Coil( #POWER_Status )
   END_RUNG
   // the same network as SCL:
   #"X-RAY_HL" := (#DATA_Generator.X_RAY_Status AND (#DATA_Generator.CMD_STAT OR "Clock_1Hz")) OR #DATA_Generator.X_RAY_Status;
   #POWER_Status := #POWER_Status AND #DATA_Generator.X_RAY_Status;
END_REGION

REGION Network 10 (SCL): Проверка ошибок от генератора
   IF #DATA_Generator.FLT[0] = TRUE
       OR #DATA_Generator.FLT[1] = TRUE
       OR #DATA_Generator.FLT[2] = TRUE
       OR #DATA_Generator.FLT[3] = TRUE
       OR #DATA_Generator.FLT[4] = TRUE
       OR #DATA_Generator.FLT[5] = TRUE
       OR #DATA_Generator.FLT[6] = TRUE
       OR #DATA_Generator.FLT[7] = TRUE
       OR #DATA_Generator.FLT[8] = TRUE
       OR #DATA_Generator.FLT[8] = TRUE
       OR #DATA_Generator.cmdError = TRUE
   THEN
       #Fault := TRUE;
   ELSE
       #Fault := FALSE;
   END_IF;
END_REGION

REGION Network 11: Проверка готовности генератора
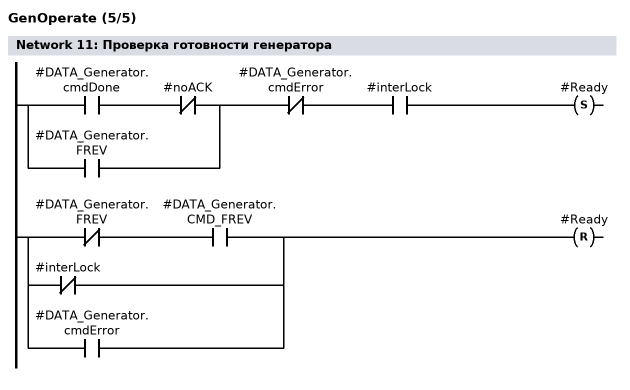
   RUNG wire#powerrail
      Contact( #DATA_Generator.cmdDone )
      I_Contact( #noACK )
      wire#w1
      I_Contact( #DATA_Generator.cmdError )
      Contact( #interLock )
      S_Coil( #Ready )
   END_RUNG
   RUNG wire#powerrail
      Contact( #DATA_Generator.FREV )
   END_RUNG wire#w1
   RUNG wire#powerrail
      I_Contact( #DATA_Generator.FREV )
      Contact( #DATA_Generator.CMD_FREV )
      wire#w2
      R_Coil( #Ready )
   END_RUNG
   RUNG wire#powerrail
      I_Contact( #interLock )
   END_RUNG wire#w2
   RUNG wire#powerrail
      Contact( #DATA_Generator.cmdError )
   END_RUNG wire#w2
   // the same network as SCL:
   IF ((#DATA_Generator.cmdDone AND NOT #noACK) OR #DATA_Generator.FREV) AND NOT #DATA_Generator.cmdError AND #interLock THEN
       #Ready := TRUE;
   END_IF;
   IF (NOT #DATA_Generator.FREV AND #DATA_Generator.CMD_FREV) OR NOT #interLock OR #DATA_Generator.cmdError THEN
       #Ready := FALSE;
   END_IF;
END_REGION

REGION Network 12 (SCL)
   #Status := #DATA_Generator.cmdState;
END_REGION
END_FUNCTION_BLOCK

FUNCTION "CheckPresset" : Void   // FC1, SCL
{ S7_Optimized_Access := 'TRUE' }
VERSION : 0.1
   VAR_INPUT
      VP_max_kV : Real;
      VP_min_kV : Real;
      CP_max_uA : UInt;
      CP_min_uA : UInt;
      "FEED_max_%" : UInt;
      "FEED_min_%" : UInt;
   END_VAR
   VAR_OUTPUT
      error : Bool;
   END_VAR
   VAR_IN_OUT
      DATA_MIDLE : "typePresset";
      DATA_LOW : "typePresset";
      DATA_HIGH : "typePresset";
   END_VAR
   VAR_TEMP
      error_check : Bool;
   END_VAR
BEGIN
   #error_check := TRUE;
   // Проверка диапазона напряжений МАКСИМУМ
   IF #DATA_LOW.VP > #VP_max_kV THEN
       // Statement section IF
       #DATA_LOW.VP := #VP_max_kV;
   ELSE
       #error_check := FALSE;
   END_IF;

   IF #DATA_MIDLE.VP > #VP_max_kV THEN
       // Statement section IF
       #DATA_MIDLE.VP := #VP_max_kV;
   ELSE
       #error_check := FALSE;
   END_IF;

   IF #DATA_HIGH.VP > #VP_max_kV THEN
       // Statement section IF
       #DATA_HIGH.VP := #VP_max_kV;
   ELSE
       #error_check := FALSE;
   END_IF;

   // Проверка диапазона напряжений МИНИМУМ
   IF #DATA_LOW.VP < #VP_min_kV THEN
       // Statement section IF
       #DATA_LOW.VP := #VP_min_kV;
   ELSE
       #error_check := FALSE;
   END_IF;

   IF #DATA_MIDLE.VP < #VP_min_kV THEN
       // Statement section IF
       #DATA_MIDLE.VP := #VP_min_kV;
   ELSE
       #error_check := FALSE;
   END_IF;

   IF #DATA_HIGH.VP < #VP_min_kV THEN
       // Statement section IF
       #DATA_HIGH.VP := #VP_min_kV;
   ELSE
       #error_check := FALSE;
   END_IF;

   // Проверка диапазона токов МАКСИМУМ
   IF #DATA_LOW.CP > #CP_max_uA THEN
       // Statement section IF
       #DATA_LOW.CP := #CP_max_uA;
   ELSE
       #error_check := FALSE;
   END_IF;

   IF #DATA_MIDLE.CP > #CP_max_uA THEN
       // Statement section IF
       #DATA_MIDLE.CP := #CP_max_uA;
   ELSE
       #error_check := FALSE;
   END_IF;

   IF #DATA_HIGH.CP > #CP_max_uA THEN
       // Statement section IF
       #DATA_HIGH.CP := #CP_max_uA;
   ELSE
       #error_check := FALSE;
   END_IF;

   // Проверка диапазона токов МИНИМУМ
   IF #DATA_LOW.CP < #CP_min_uA THEN
       // Statement section IF
       #DATA_LOW.CP := #CP_min_uA;
   ELSE
       #error_check := FALSE;
   END_IF;

   IF #DATA_MIDLE.CP < #CP_min_uA THEN
       // Statement section IF
       #DATA_MIDLE.CP := #CP_min_uA;
   ELSE
       #error_check := FALSE;
   END_IF;

   IF #DATA_HIGH.CP < #CP_min_uA THEN
       // Statement section IF
       #DATA_HIGH.CP := #CP_min_uA;
   ELSE
       #error_check := FALSE;
   END_IF;

   // Проверка диапазона скорости шторки МАКСИМУМ
   IF #DATA_LOW.Velocity > #"FEED_max_%" THEN
       // Statement section IF
       #DATA_LOW.Velocity := #"FEED_max_%";
   ELSE
       #error_check := FALSE;
   END_IF;


   IF #DATA_MIDLE.Velocity > #"FEED_max_%" THEN
       // Statement section IF
       #DATA_MIDLE.Velocity := #"FEED_max_%";
   ELSE
       #error_check := FALSE;
   END_IF;

   IF #DATA_HIGH.Velocity > #"FEED_max_%" THEN
       // Statement section IF
       #DATA_HIGH.Velocity := #"FEED_max_%";
   ELSE
       #error_check := FALSE;
   END_IF;

   // Проверка диапазона скорости шторки МИНИМУМ
   IF #DATA_LOW.Velocity < #"FEED_min_%" THEN
       // Statement section IF
       #DATA_LOW.Velocity := #"FEED_min_%";
   ELSE
       #error_check := FALSE;
   END_IF;


   IF #DATA_MIDLE.Velocity < #"FEED_min_%" THEN
       // Statement section IF
       #DATA_MIDLE.Velocity := #"FEED_min_%";
   ELSE
       #error_check := FALSE;
   END_IF;

   IF #DATA_HIGH.Velocity < #"FEED_min_%" THEN
       // Statement section IF
       #DATA_HIGH.Velocity := #"FEED_min_%";
   ELSE
       #error_check := FALSE;
   END_IF;

   #error := #error_check;
END_FUNCTION

FUNCTION "CHeckVpCp" : Void   // FC3, SCL
{ S7_Optimized_Access := 'TRUE' }
VERSION : 0.1
   VAR_INPUT
      VP_set : Real;
      CP_set : UInt;
      VP_monitor : Real;
      CP_monitor : Real;
      Tolerance_Vp_kV : Real;
      Tolerance_CP_uA : Real;
   END_VAR
   VAR_OUTPUT
      Value_EQ : Bool;
      Delta_VP : Real;
      Delta_CP : Real;
   END_VAR
   VAR_TEMP
      DeltaVP : Real;
      DeltaCP : Real;
   END_VAR
BEGIN
   #DeltaVP := ABS(#VP_set - #VP_monitor);
   #DeltaCP := ABS(#CP_set - #CP_monitor);

   IF #VP_set = 0.0 OR #CP_set = 0 THEN
       #Value_EQ := FALSE;
       RETURN;
   END_IF;

   IF (#DeltaVP < #Tolerance_Vp_kV) AND (#DeltaCP < #Tolerance_CP_uA) THEN
       // Statement section IF
       #Value_EQ:=TRUE;
   ELSE
       #Value_EQ := FALSE;
   END_IF;

   #Delta_VP := #DeltaVP;
   #Delta_CP := #DeltaCP;
END_FUNCTION

FUNCTION "LoadPresset" : Void   // FC4, SCL
{ S7_Optimized_Access := 'TRUE' }
VERSION : 0.1
   VAR_INPUT
      N_Presset : UInt;
      DATA_from : "typePresset";
   END_VAR
   VAR_OUTPUT
      DATA_to : "typeGeneratorDATA";
   END_VAR
BEGIN
   #DATA_to.VP_Programm := #DATA_from.VP;
   #DATA_to.CP_Programm := #DATA_from.CP;
END_FUNCTION

FUNCTION "GeneratorStage" : Void   // FC9, LAD
{ S7_Optimized_Access := 'TRUE' }
VERSION : 0.1
   VAR_IN_OUT
      DATA_Generator1 : "typeGeneratorDATA";
      DATA_Generator2 : "typeGeneratorDATA";
   END_VAR
   VAR_TEMP
      err_Check_Presset : Bool;
      HL_XRAY_1 : Bool;
      HL_XRAY_2 : Bool;
   END_VAR
BEGIN

REGION Network 1: Проверка уставок
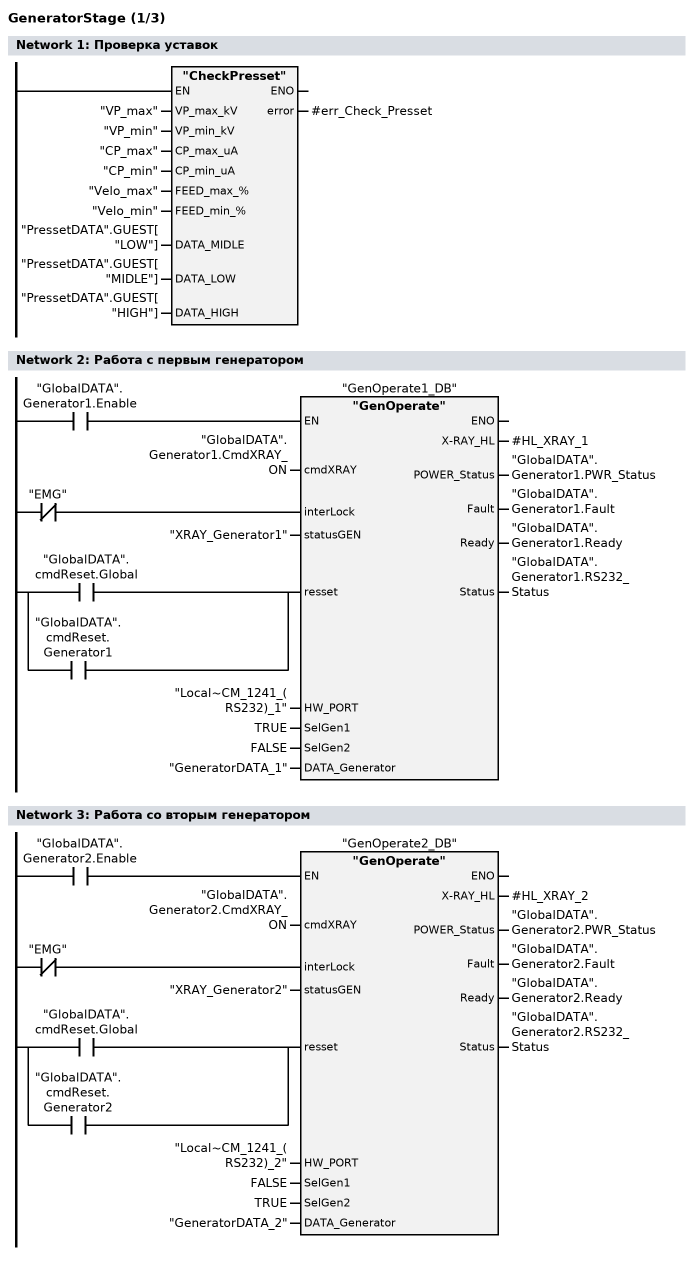
   RUNG wire#powerrail
      "CheckPresset"(VP_max_kV := "VP_max", VP_min_kV := "VP_min", CP_max_uA := "CP_max", CP_min_uA := "CP_min", "FEED_max_%" := "Velo_max", "FEED_min_%" := "Velo_min", DATA_MIDLE := "PressetDATA".GUEST["LOW"], DATA_LOW := "PressetDATA".GUEST["MIDLE"], DATA_HIGH := "PressetDATA".GUEST["HIGH"], error => #err_Check_Presset)
   END_RUNG
   // the same network as SCL:
   "CheckPresset"(VP_max_kV := "VP_max",
                  VP_min_kV := "VP_min",
                  CP_max_uA := "CP_max",
                  CP_min_uA := "CP_min",
                  "FEED_max_%" := "Velo_max",
                  "FEED_min_%" := "Velo_min",
                  DATA_MIDLE := "PressetDATA".GUEST["LOW"],
                  DATA_LOW := "PressetDATA".GUEST["MIDLE"],
                  DATA_HIGH := "PressetDATA".GUEST["HIGH"],
                  error => #err_Check_Presset);
END_REGION

REGION Network 2: Работа с первым генератором
   RUNG wire#powerrail
      Contact( "GlobalDATA".Generator1.Enable )
      "GenOperate1_DB"(interLock := wire#w1, resset := wire#w2, cmdXRAY := "GlobalDATA".Generator1.CmdXRAY_ON, statusGEN := "XRAY_Generator1", HW_PORT := "Local~CM_1241_(RS232)_1", SelGen1 := TRUE, SelGen2 := FALSE, DATA_Generator := "GeneratorDATA_1", "X-RAY_HL" => #HL_XRAY_1, POWER_Status => "GlobalDATA".Generator1.PWR_Status, Fault => "GlobalDATA".Generator1.Fault, Ready => "GlobalDATA".Generator1.Ready, Status => "GlobalDATA".Generator1.RS232_Status)
   END_RUNG
   RUNG wire#powerrail
      I_Contact( "EMG" )
   END_RUNG wire#w1
   RUNG wire#powerrail
      Contact( "GlobalDATA".cmdReset.Global )
   END_RUNG wire#w2
   RUNG wire#powerrail
      Contact( "GlobalDATA".cmdReset.Generator1 )
   END_RUNG wire#w2
   // the same network as SCL:
   IF "GlobalDATA".Generator1.Enable THEN
       "GenOperate1_DB"(cmdXRAY := "GlobalDATA".Generator1.CmdXRAY_ON,   // "GenOperate"
                        interLock := NOT "EMG",
                        statusGEN := "XRAY_Generator1",
                        resset := "GlobalDATA".cmdReset.Global OR "GlobalDATA".cmdReset.Generator1,
                        HW_PORT := "Local~CM_1241_(RS232)_1",
                        SelGen1 := TRUE,
                        SelGen2 := FALSE,
                        DATA_Generator := "GeneratorDATA_1",
                        "X-RAY_HL" => #HL_XRAY_1,
                        POWER_Status => "GlobalDATA".Generator1.PWR_Status,
                        Fault => "GlobalDATA".Generator1.Fault,
                        Ready => "GlobalDATA".Generator1.Ready,
                        Status => "GlobalDATA".Generator1.RS232_Status);
   END_IF;
END_REGION

REGION Network 3: Работа со вторым генератором
   RUNG wire#powerrail
      Contact( "GlobalDATA".Generator2.Enable )
      "GenOperate2_DB"(interLock := wire#w1, resset := wire#w2, cmdXRAY := "GlobalDATA".Generator2.CmdXRAY_ON, statusGEN := "XRAY_Generator2", HW_PORT := "Local~CM_1241_(RS232)_2", SelGen1 := FALSE, SelGen2 := TRUE, DATA_Generator := "GeneratorDATA_2", "X-RAY_HL" => #HL_XRAY_2, POWER_Status => "GlobalDATA".Generator2.PWR_Status, Fault => "GlobalDATA".Generator2.Fault, Ready => "GlobalDATA".Generator2.Ready, Status => "GlobalDATA".Generator2.RS232_Status)
   END_RUNG
   RUNG wire#powerrail
      I_Contact( "EMG" )
   END_RUNG wire#w1
   RUNG wire#powerrail
      Contact( "GlobalDATA".cmdReset.Global )
   END_RUNG wire#w2
   RUNG wire#powerrail
      Contact( "GlobalDATA".cmdReset.Generator2 )
   END_RUNG wire#w2
   // the same network as SCL:
   IF "GlobalDATA".Generator2.Enable THEN
       "GenOperate2_DB"(cmdXRAY := "GlobalDATA".Generator2.CmdXRAY_ON,   // "GenOperate"
                        interLock := NOT "EMG",
                        statusGEN := "XRAY_Generator2",
                        resset := "GlobalDATA".cmdReset.Global OR "GlobalDATA".cmdReset.Generator2,
                        HW_PORT := "Local~CM_1241_(RS232)_2",
                        SelGen1 := FALSE,
                        SelGen2 := TRUE,
                        DATA_Generator := "GeneratorDATA_2",
                        "X-RAY_HL" => #HL_XRAY_2,
                        POWER_Status => "GlobalDATA".Generator2.PWR_Status,
                        Fault => "GlobalDATA".Generator2.Fault,
                        Ready => "GlobalDATA".Generator2.Ready,
                        Status => "GlobalDATA".Generator2.RS232_Status);
   END_IF;
END_REGION

REGION Network 4 (SCL): Передача в глобальный блок данных состояния генератора 1
   "GlobalDATA".Generator1.CP_monitor := #DATA_Generator1.CP_Monitor;
   "GlobalDATA".Generator1.VP_monitor := #DATA_Generator1.VP_Monitor;
   "GlobalDATA".Generator1.T_monitor := #DATA_Generator1.T_Monitor;
   "GlobalDATA".Generator1.CP := #DATA_Generator1.CP_Programm;
   "GlobalDATA".Generator1.VP := #DATA_Generator1.VP_Programm;
   "GlobalDATA".Generator1.XRAY_Status := #DATA_Generator1.X_RAY_Status;
   "GlobalDATA".Generator1.FLT[0] := #DATA_Generator1.FLT[0];
   "GlobalDATA".Generator1.FLT[1] := #DATA_Generator1.FLT[1];
   "GlobalDATA".Generator1.FLT[2] := #DATA_Generator1.FLT[2];
   "GlobalDATA".Generator1.FLT[3] := #DATA_Generator1.FLT[3];
   "GlobalDATA".Generator1.FLT[4] := #DATA_Generator1.FLT[4];
   "GlobalDATA".Generator1.FLT[5] := #DATA_Generator1.FLT[5];
   "GlobalDATA".Generator1.FLT[6] := #DATA_Generator1.FLT[6];
   "GlobalDATA".Generator1.FLT[7] := #DATA_Generator1.FLT[7];
   "GlobalDATA".Generator1.FLT[8] := #DATA_Generator1.FLT[8];
   "GlobalDATA".Generator1.FLT[9] := #DATA_Generator1.FLT[9];
END_REGION

REGION Network 5 (SCL): Передача в глобальный блок данных состояния генератора 2
   "GlobalDATA".Generator2.CP_monitor := #DATA_Generator2.CP_Monitor;
   "GlobalDATA".Generator2.VP_monitor := #DATA_Generator2.VP_Monitor;
   "GlobalDATA".Generator2.T_monitor := #DATA_Generator2.T_Monitor;
   "GlobalDATA".Generator2.CP := #DATA_Generator2.CP_Programm;
   "GlobalDATA".Generator2.VP := #DATA_Generator2.VP_Programm;
   "GlobalDATA".Generator2.FLT[0] := #DATA_Generator2.FLT[0];
   "GlobalDATA".Generator2.FLT[1] := #DATA_Generator2.FLT[1];
   "GlobalDATA".Generator2.FLT[2] := #DATA_Generator2.FLT[2];
   "GlobalDATA".Generator2.FLT[3] := #DATA_Generator2.FLT[3];
   "GlobalDATA".Generator2.FLT[4] := #DATA_Generator2.FLT[4];
   "GlobalDATA".Generator2.FLT[5] := #DATA_Generator2.FLT[5];
   "GlobalDATA".Generator2.FLT[6] := #DATA_Generator2.FLT[6];
   "GlobalDATA".Generator2.FLT[7] := #DATA_Generator2.FLT[7];
   "GlobalDATA".Generator2.FLT[8] := #DATA_Generator2.FLT[8];
   "GlobalDATA".Generator2.FLT[9] := #DATA_Generator2.FLT[9];
END_REGION

REGION Network 6: Relay switch OFF Fun Generator 2
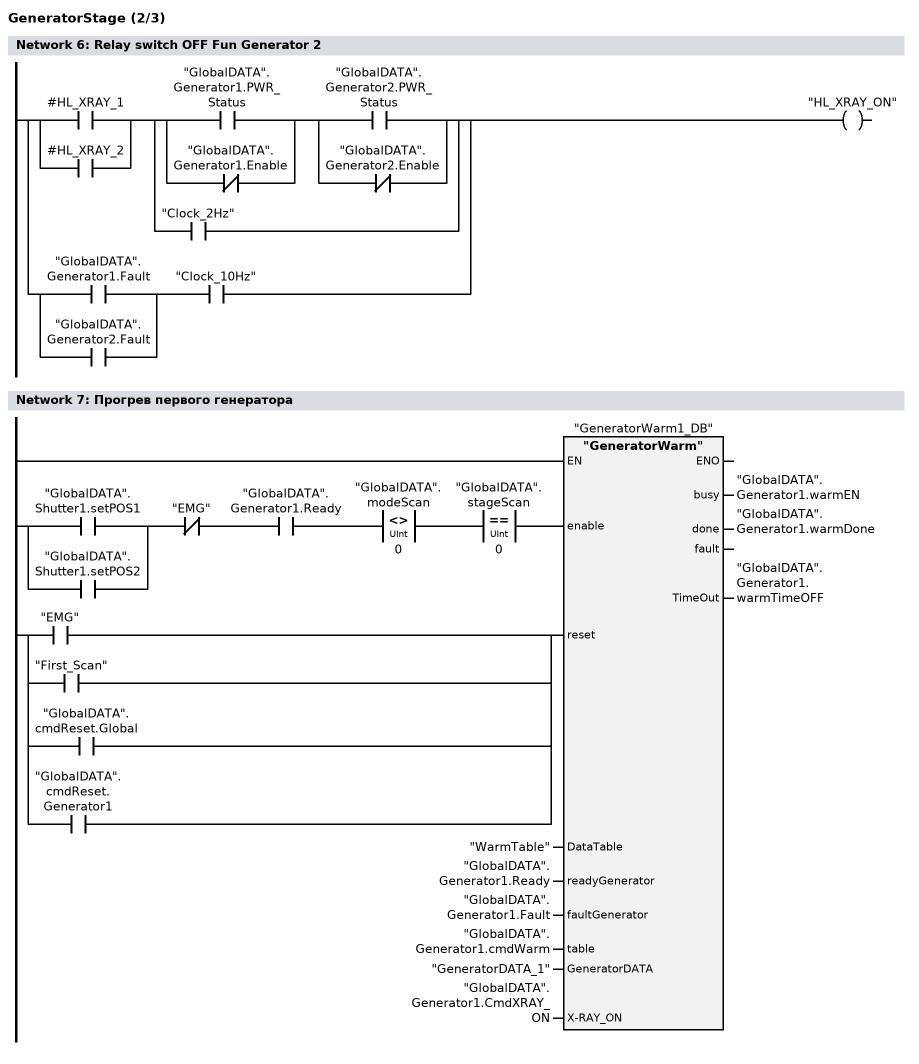
   RUNG wire#powerrail
      Contact( #HL_XRAY_1 )
      wire#w1
      Contact( "GlobalDATA".Generator1.PWR_Status )
      wire#w2
      Contact( "GlobalDATA".Generator2.PWR_Status )
      wire#w3
      Coil( "HL_XRAY_ON" )
   END_RUNG
   RUNG wire#powerrail
      Contact( #HL_XRAY_2 )
   END_RUNG wire#w1
   RUNG wire#w1
      I_Contact( "GlobalDATA".Generator1.Enable )
   END_RUNG wire#w2
   RUNG wire#w2
      I_Contact( "GlobalDATA".Generator2.Enable )
   END_RUNG wire#w3
   RUNG wire#w1
      Contact( "Clock_2Hz" )
   END_RUNG wire#w3
   RUNG wire#powerrail
      Contact( "GlobalDATA".Generator1.Fault )
      wire#w4
      Contact( "Clock_10Hz" )
   END_RUNG wire#w3
   RUNG wire#powerrail
      Contact( "GlobalDATA".Generator2.Fault )
   END_RUNG wire#w4
   // the same network as SCL:
   "HL_XRAY_ON" := ((#HL_XRAY_1 OR #HL_XRAY_2) AND ((("GlobalDATA".Generator1.PWR_Status OR NOT "GlobalDATA".Generator1.Enable) AND ("GlobalDATA".Generator2.PWR_Status OR NOT "GlobalDATA".Generator2.Enable)) OR "Clock_2Hz")) OR (("GlobalDATA".Generator1.Fault OR "GlobalDATA".Generator2.Fault) AND "Clock_10Hz");
END_REGION

REGION Network 7: Прогрев первого генератора
   RUNG wire#powerrail
      "GeneratorWarm1_DB"(enable := wire#w2, reset := wire#w3, DataTable := "WarmTable", readyGenerator := "GlobalDATA".Generator1.Ready, faultGenerator := "GlobalDATA".Generator1.Fault, table := "GlobalDATA".Generator1.cmdWarm, GeneratorDATA := "GeneratorDATA_1", "X-RAY_ON" := "GlobalDATA".Generator1.CmdXRAY_ON, busy => "GlobalDATA".Generator1.warmEN, done => "GlobalDATA".Generator1.warmDone, fault =>, TimeOut => "GlobalDATA".Generator1.warmTimeOFF)
   END_RUNG
   RUNG wire#powerrail
      Contact( "GlobalDATA".Shutter1.setPOS1 )
      wire#w1
      I_Contact( "EMG" )
      Contact( "GlobalDATA".Generator1.Ready )
      { S7_Templates := "SrcType := UInt" } NE_Contact(in1 := "GlobalDATA".modeScan, in2 := 0)
      { S7_Templates := "SrcType := UInt" } EQ_Contact(in1 := "GlobalDATA".stageScan, in2 := 0)
   END_RUNG wire#w2
   RUNG wire#powerrail
      Contact( "GlobalDATA".Shutter1.setPOS2 )
   END_RUNG wire#w1
   RUNG wire#powerrail
      Contact( "EMG" )
   END_RUNG wire#w3
   RUNG wire#powerrail
      Contact( "First_Scan" )
   END_RUNG wire#w3
   RUNG wire#powerrail
      Contact( "GlobalDATA".cmdReset.Global )
   END_RUNG wire#w3
   RUNG wire#powerrail
      Contact( "GlobalDATA".cmdReset.Generator1 )
   END_RUNG wire#w3
   // the same network as SCL:
   "GeneratorWarm1_DB"(enable := ("GlobalDATA".Shutter1.setPOS1 OR "GlobalDATA".Shutter1.setPOS2) AND NOT "EMG" AND "GlobalDATA".Generator1.Ready AND ("GlobalDATA".modeScan <> 0) AND ("GlobalDATA".stageScan = 0),   // "GeneratorWarm"
                       reset := "EMG" OR "First_Scan" OR "GlobalDATA".cmdReset.Global OR "GlobalDATA".cmdReset.Generator1,
                       DataTable := "WarmTable",
                       readyGenerator := "GlobalDATA".Generator1.Ready,
                       faultGenerator := "GlobalDATA".Generator1.Fault,
                       table := "GlobalDATA".Generator1.cmdWarm,
                       GeneratorDATA := "GeneratorDATA_1",
                       "X-RAY_ON" := "GlobalDATA".Generator1.CmdXRAY_ON,
                       busy => "GlobalDATA".Generator1.warmEN,
                       done => "GlobalDATA".Generator1.warmDone,
                       TimeOut => "GlobalDATA".Generator1.warmTimeOFF);
END_REGION

REGION Network 8: Прогрев второго генератора
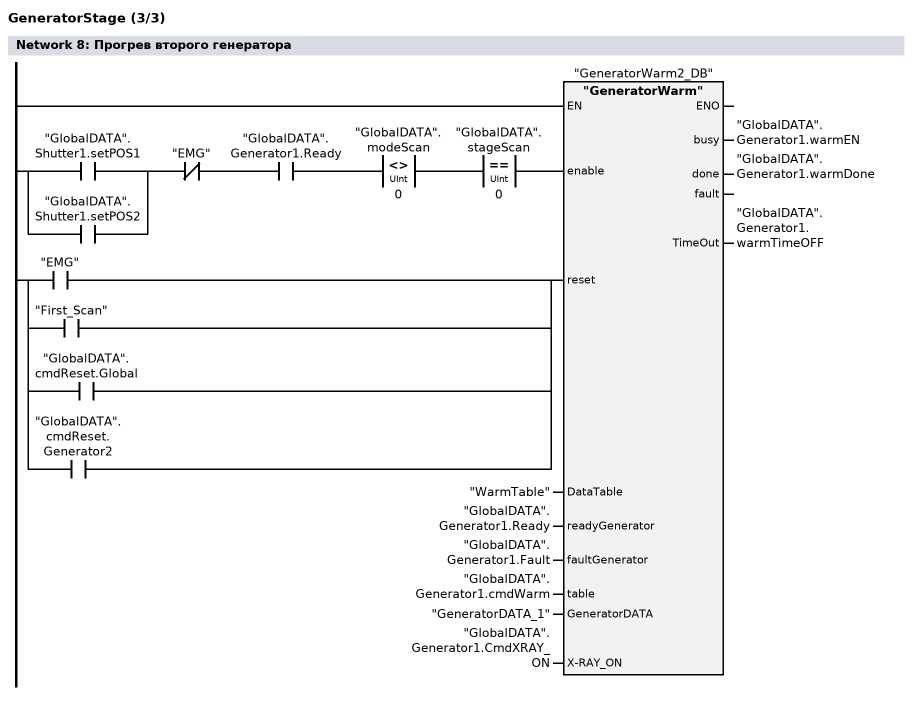
   RUNG wire#powerrail
      "GeneratorWarm2_DB"(enable := wire#w2, reset := wire#w3, DataTable := "WarmTable", readyGenerator := "GlobalDATA".Generator1.Ready, faultGenerator := "GlobalDATA".Generator1.Fault, table := "GlobalDATA".Generator1.cmdWarm, GeneratorDATA := "GeneratorDATA_1", "X-RAY_ON" := "GlobalDATA".Generator1.CmdXRAY_ON, busy => "GlobalDATA".Generator1.warmEN, done => "GlobalDATA".Generator1.warmDone, fault =>, TimeOut => "GlobalDATA".Generator1.warmTimeOFF)
   END_RUNG
   RUNG wire#powerrail
      Contact( "GlobalDATA".Shutter1.setPOS1 )
      wire#w1
      I_Contact( "EMG" )
      Contact( "GlobalDATA".Generator1.Ready )
      { S7_Templates := "SrcType := UInt" } NE_Contact(in1 := "GlobalDATA".modeScan, in2 := 0)
      { S7_Templates := "SrcType := UInt" } EQ_Contact(in1 := "GlobalDATA".stageScan, in2 := 0)
   END_RUNG wire#w2
   RUNG wire#powerrail
      Contact( "GlobalDATA".Shutter1.setPOS2 )
   END_RUNG wire#w1
   RUNG wire#powerrail
      Contact( "EMG" )
   END_RUNG wire#w3
   RUNG wire#powerrail
      Contact( "First_Scan" )
   END_RUNG wire#w3
   RUNG wire#powerrail
      Contact( "GlobalDATA".cmdReset.Global )
   END_RUNG wire#w3
   RUNG wire#powerrail
      Contact( "GlobalDATA".cmdReset.Generator2 )
   END_RUNG wire#w3
   // the same network as SCL:
   "GeneratorWarm2_DB"(enable := ("GlobalDATA".Shutter1.setPOS1 OR "GlobalDATA".Shutter1.setPOS2) AND NOT "EMG" AND "GlobalDATA".Generator1.Ready AND ("GlobalDATA".modeScan <> 0) AND ("GlobalDATA".stageScan = 0),   // "GeneratorWarm"
                       reset := "EMG" OR "First_Scan" OR "GlobalDATA".cmdReset.Global OR "GlobalDATA".cmdReset.Generator2,
                       DataTable := "WarmTable",
                       readyGenerator := "GlobalDATA".Generator1.Ready,
                       faultGenerator := "GlobalDATA".Generator1.Fault,
                       table := "GlobalDATA".Generator1.cmdWarm,
                       GeneratorDATA := "GeneratorDATA_1",
                       "X-RAY_ON" := "GlobalDATA".Generator1.CmdXRAY_ON,
                       busy => "GlobalDATA".Generator1.warmEN,
                       done => "GlobalDATA".Generator1.warmDone,
                       TimeOut => "GlobalDATA".Generator1.warmTimeOFF);
END_REGION
END_FUNCTION

// folder: IR

ORGANIZATION_BLOCK "IR1 Faling HW Int"   // OB40, SCL, HWProcessInterrupt
{ S7_Optimized_Access := 'TRUE' }
VERSION : 0.1
   VAR_INPUT
      LADDR : Hw_Io;   // Hardware identifier
      USI : Word;   // User structure identifier
      IChannel : USInt;   // Interrupt channel number
      EventType : Byte;   // EventType
   END_VAR
   VAR_TEMP
      retval : Int;
   END_VAR
BEGIN
   #retval := RD_SYS_T("IR".IR1_t2);
   "IR".Guest["IR".Guest_index].IR1["IR".IR1_count].t2:= "IR".IR1_t2;
   "IR".Guest["IR".Guest_index].IR1["IR".IR1_count].delta := T_DIFF(IN1 := "IR".Guest["IR".Guest_index].IR1["IR".IR1_count].t2, IN2 := "IR".Guest["IR".Guest_index].IR1["IR".IR1_count].t1);


   "IR".IR1_count := "IR".IR1_count + 1;
   "IR".Guest["IR".Guest_index].count := "IR".IR1_count;
   IF "IR".IR1_count > 4 THEN
       "IR".IR1_count := 0;
   END_IF;

   //"HL1" := 0;
END_ORGANIZATION_BLOCK

ORGANIZATION_BLOCK "IR1 Rising HW Int"   // OB41, SCL, HWProcessInterrupt
{ S7_Optimized_Access := 'TRUE' }
VERSION : 0.1
   VAR_INPUT
      LADDR : Hw_Io;   // Hardware identifier
      USI : Word;   // User structure identifier
      IChannel : USInt;   // Interrupt channel number
      EventType : Byte;   // EventType
   END_VAR
   VAR_TEMP
      retval : Int;
   END_VAR
BEGIN
   IF ("IR".Guest_came = 0) THEN
       #retval := RD_SYS_T("IR".IR1_t1);
       "IR".Guest["IR".Guest_index].IR1_t1 := "IR".IR1_t1;
       "IR".Guest["IR".Guest_index].IR1["IR".IR1_count].t1 := "IR".IR1_t1;
       "IR".Guest_came := 1;
   ELSE
       #retval := RD_SYS_T("IR".Guest["IR".Guest_index].IR1["IR".IR1_count].t1);
   END_IF;


   //"HL1" := 1;
END_ORGANIZATION_BLOCK

ORGANIZATION_BLOCK "IR2 Faling HW Int"   // OB42, SCL, HWProcessInterrupt
{ S7_Optimized_Access := 'TRUE' }
VERSION : 0.1
   VAR_INPUT
      LADDR : Hw_Io;   // Hardware identifier
      USI : Word;   // User structure identifier
      IChannel : USInt;   // Interrupt channel number
      EventType : Byte;   // EventType
   END_VAR
   VAR_TEMP
      retval : Int;
   END_VAR
BEGIN
   IF "IR".Guest_came = 1 THEN

       ;
   END_IF;
END_ORGANIZATION_BLOCK

ORGANIZATION_BLOCK "IR2 Rising HW Int"   // OB43, SCL, HWProcessInterrupt
{ S7_Optimized_Access := 'TRUE' }
VERSION : 0.1
   VAR_INPUT
      LADDR : Hw_Io;   // Hardware identifier
      USI : Word;   // User structure identifier
      IChannel : USInt;   // Interrupt channel number
      EventType : Byte;   // EventType
   END_VAR
   VAR_TEMP
      retval : Int;
   END_VAR
BEGIN
   IF "IR".Guest_came = 1 AND  "IR".SHOT_make = 0 THEN
       #retval := RD_SYS_T("IR".IR2_t1);

       "IR".Guest["IR".Guest_index].IR2_t1 := "IR".IR2_t1;
       "IR".Delta_IR2_IR1 := T_DIFF(IN1 := "IR".IR2_t1, IN2 := "IR".IR1_t1);
       "IR".Guest["IR".Guest_index].Delta_IR2_IR1 := "IR".Delta_IR2_IR1;

       "IR".IR1_count := 0;
       "IR".SHOT_make := 1;

       "IR".Guest_index := "IR".Guest_index + 1;
       IF "IR".Guest_index > 99 THEN
           "IR".Guest_index := 0;
       END_IF;
   END_IF;
END_ORGANIZATION_BLOCK

ORGANIZATION_BLOCK "Rising_X-RAY"   // OB44, SCL, HWProcessInterrupt
{ S7_Optimized_Access := 'TRUE' }
VERSION : 0.1
   VAR_INPUT
      LADDR : Hw_Io;   // Hardware identifier
      USI : Word;   // User structure identifier
      IChannel : USInt;   // Interrupt channel number
      EventType : Byte;   // EventType
   END_VAR
   VAR_TEMP
      retval : Int;
   END_VAR
BEGIN
   #retval := RD_SYS_T("temp"."T1_X-RAY");
   "HL_XRAY_ON" := TRUE;
END_ORGANIZATION_BLOCK

ORGANIZATION_BLOCK "Falling_X-RAY"   // OB45, SCL, HWProcessInterrupt
{ S7_Optimized_Access := 'TRUE' }
VERSION : 0.1
   VAR_INPUT
      LADDR : Hw_Io;   // Hardware identifier
      USI : Word;   // User structure identifier
      IChannel : USInt;   // Interrupt channel number
      EventType : Byte;   // EventType
   END_VAR
   VAR_TEMP
      retval : Int;
   END_VAR
BEGIN
   #retval := RD_SYS_T("temp"."T2_X-RAY");

   "temp".T_XRAY:= T_DIFF(IN1 := "temp"."T2_X-RAY", IN2 := "temp"."T1_X-RAY");

   "HL_XRAY_ON" := FALSE;
END_ORGANIZATION_BLOCK

// folder: Power&Reset

FUNCTION "ResetManagment" : Void   // FC10, LAD
{ S7_Optimized_Access := 'TRUE' }
VERSION : 0.1
BEGIN

REGION Network 1: Формирование импульса сброса
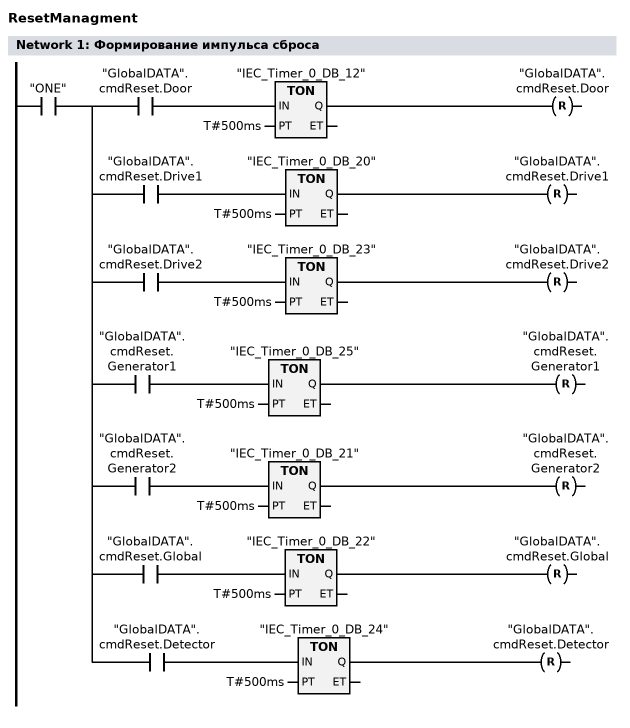
   "IEC_Timer_0_DB_12".TON(IN := "ONE" AND "GlobalDATA".cmdReset.Door, PT := T#500ms);
   IF "IEC_Timer_0_DB_12".Q THEN "GlobalDATA".cmdReset.Door := FALSE; END_IF;
   "IEC_Timer_0_DB_20".TON(IN := "ONE" AND "GlobalDATA".cmdReset.Drive1, PT := T#500ms);
   IF "IEC_Timer_0_DB_20".Q THEN "GlobalDATA".cmdReset.Drive1 := FALSE; END_IF;
   "IEC_Timer_0_DB_23".TON(IN := "ONE" AND "GlobalDATA".cmdReset.Drive2, PT := T#500ms);
   IF "IEC_Timer_0_DB_23".Q THEN "GlobalDATA".cmdReset.Drive2 := FALSE; END_IF;
   "IEC_Timer_0_DB_25".TON(IN := "ONE" AND "GlobalDATA".cmdReset.Generator1, PT := T#500ms);
   IF "IEC_Timer_0_DB_25".Q THEN "GlobalDATA".cmdReset.Generator1 := FALSE; END_IF;
   "IEC_Timer_0_DB_21".TON(IN := "ONE" AND "GlobalDATA".cmdReset.Generator2, PT := T#500ms);
   IF "IEC_Timer_0_DB_21".Q THEN "GlobalDATA".cmdReset.Generator2 := FALSE; END_IF;
   "IEC_Timer_0_DB_22".TON(IN := "ONE" AND "GlobalDATA".cmdReset.Global, PT := T#500ms);
   IF "IEC_Timer_0_DB_22".Q THEN "GlobalDATA".cmdReset.Global := FALSE; END_IF;
   "IEC_Timer_0_DB_24".TON(IN := "ONE" AND "GlobalDATA".cmdReset.Detector, PT := T#500ms);
   IF "IEC_Timer_0_DB_24".Q THEN "GlobalDATA".cmdReset.Detector := FALSE; END_IF;
END_REGION
END_FUNCTION

FUNCTION "PowerManagment" : Void   // FC11, LAD
{ S7_Optimized_Access := 'TRUE' }
VERSION : 0.1
BEGIN

REGION Network 1 (SCL): Проверка ошибок по пускателю или автоматическим выключателям
   // Если нет ошибок по пускателям и автоматам, то даем команду на включение пускателя
   // Если выбран режим где включено оборудование
   IF "GlobalDATA".modeScan = "modeAUTO" OR "GlobalDATA".modeScan = "modeJOG" OR "GlobalDATA".modeScan = "modeSERVIСE" THEN
       //Генератор 1. Если нет ошибок по включению питания, то включить пускатель. Ошибки по пускателю и автоматическому выключателю
       IF "GlobalDATA".Generator1.PowerFail = FALSE THEN
           "KM_Generator1" := TRUE;
       END_IF;
       //Генератор 2. Если нет ошибок по включению питания, то включить пускатель. Ошибки по пускателю и автоматическому выключателю
       IF "GlobalDATA".Generator2.PowerFail = FALSE THEN
           "KM_Generator2" := TRUE;
       END_IF;
       //Привод двери. Если нет ошибок по включению питания, то включить пускатель. Ошибки по пускателю и автоматическому выключателю
       IF "GlobalDATA".Door.PowerFail = FALSE THEN
           "KM_Drive_Door" := TRUE;
       END_IF;
       //Питание детекторов. Если нет ошибок по включению питания, то включить пускатель. Ошибки по пускателю и автоматическому выключателю
       IF "GlobalDATA".Detector.PowerFail = FALSE THEN
           "KM_Detectors" := TRUE;
       END_IF;
   END_IF;

   //Если есть ошибки по питанию, то переводим режим в выключено. После квитирования ошибки нужно будет перевести заново в нужный режим
   IF "GlobalDATA".Generator1.PowerFail
       AND "GlobalDATA".Generator2.PowerFail
       AND "GlobalDATA".Door.PowerFail
       AND "GlobalDATA".Detector.PowerFail
   THEN
       "GlobalDATA".modeScan := "modeOFF";
   END_IF;
END_REGION

REGION Network 2: Контроль пускателей и автоматов
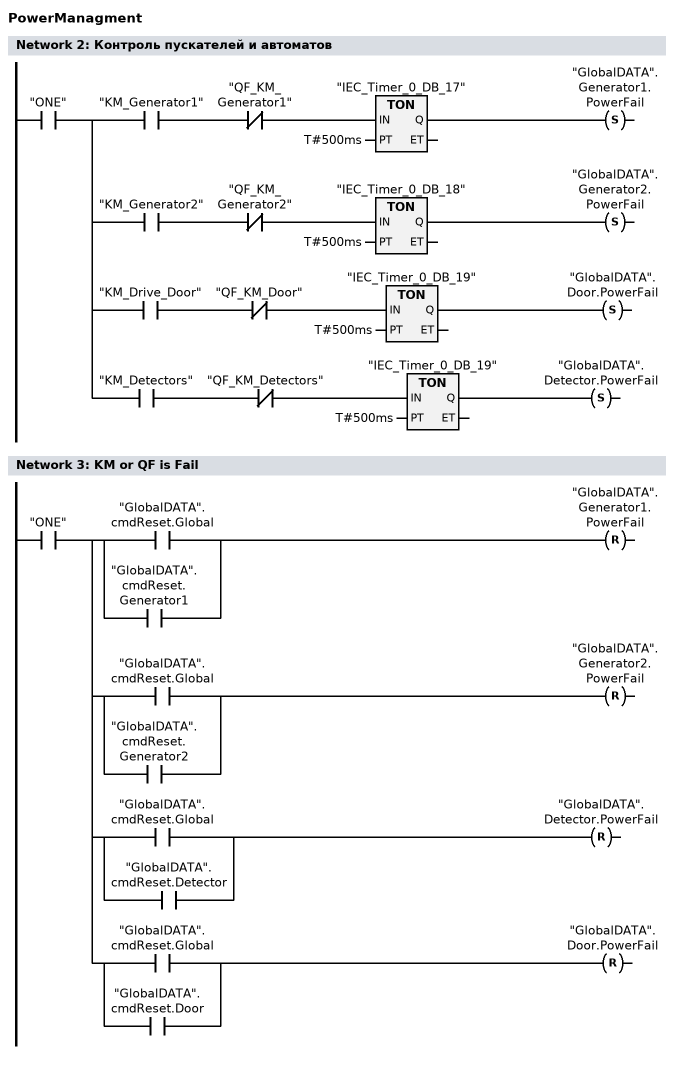
   "IEC_Timer_0_DB_17".TON(IN := "ONE" AND "KM_Generator1" AND NOT "QF_KM_Generator1", PT := T#500ms);
   IF "IEC_Timer_0_DB_17".Q THEN "GlobalDATA".Generator1.PowerFail := TRUE; END_IF;
   "IEC_Timer_0_DB_18".TON(IN := "ONE" AND "KM_Generator2" AND NOT "QF_KM_Generator2", PT := T#500ms);
   IF "IEC_Timer_0_DB_18".Q THEN "GlobalDATA".Generator2.PowerFail := TRUE; END_IF;
   "IEC_Timer_0_DB_19".TON(IN := "ONE" AND "KM_Drive_Door" AND NOT "QF_KM_Door", PT := T#500ms);
   IF "IEC_Timer_0_DB_19".Q THEN "GlobalDATA".Door.PowerFail := TRUE; END_IF;
   "IEC_Timer_0_DB_19".TON(IN := "ONE" AND "KM_Detectors" AND NOT "QF_KM_Detectors", PT := T#500ms);
   IF "IEC_Timer_0_DB_19".Q THEN "GlobalDATA".Detector.PowerFail := TRUE; END_IF;
END_REGION

REGION Network 3: KM or QF is Fail
   RUNG wire#powerrail
      Contact( "ONE" )
      wire#w1
      Contact( "GlobalDATA".cmdReset.Global )
      wire#w2
      R_Coil( "GlobalDATA".Generator1.PowerFail )
   END_RUNG
   RUNG wire#w1
      Contact( "GlobalDATA".cmdReset.Generator1 )
   END_RUNG wire#w2
   RUNG wire#w1
      Contact( "GlobalDATA".cmdReset.Global )
      wire#w3
      R_Coil( "GlobalDATA".Generator2.PowerFail )
   END_RUNG
   RUNG wire#w1
      Contact( "GlobalDATA".cmdReset.Generator2 )
   END_RUNG wire#w3
   RUNG wire#w1
      Contact( "GlobalDATA".cmdReset.Global )
      wire#w4
      R_Coil( "GlobalDATA".Detector.PowerFail )
   END_RUNG
   RUNG wire#w1
      Contact( "GlobalDATA".cmdReset.Detector )
   END_RUNG wire#w4
   RUNG wire#w1
      Contact( "GlobalDATA".cmdReset.Global )
      wire#w5
      R_Coil( "GlobalDATA".Door.PowerFail )
   END_RUNG
   RUNG wire#w1
      Contact( "GlobalDATA".cmdReset.Door )
   END_RUNG wire#w5
   // the same network as SCL:
   IF "ONE" AND ("GlobalDATA".cmdReset.Global OR "GlobalDATA".cmdReset.Generator1) THEN
       "GlobalDATA".Generator1.PowerFail := FALSE;
   END_IF;
   IF "ONE" AND ("GlobalDATA".cmdReset.Global OR "GlobalDATA".cmdReset.Generator2) THEN
       "GlobalDATA".Generator2.PowerFail := FALSE;
   END_IF;
   IF "ONE" AND ("GlobalDATA".cmdReset.Global OR "GlobalDATA".cmdReset.Detector) THEN
       "GlobalDATA".Detector.PowerFail := FALSE;
   END_IF;
   IF "ONE" AND ("GlobalDATA".cmdReset.Global OR "GlobalDATA".cmdReset.Door) THEN
       "GlobalDATA".Door.PowerFail := FALSE;
   END_IF;
END_REGION
END_FUNCTION

// folder: Safety

FUNCTION_BLOCK "Safety"   // FB7, LAD
{ S7_Optimized_Access := 'TRUE' }
VERSION : 0.1
BEGIN

REGION Network 1: Отключаем X-RAY при аварийной ситуации
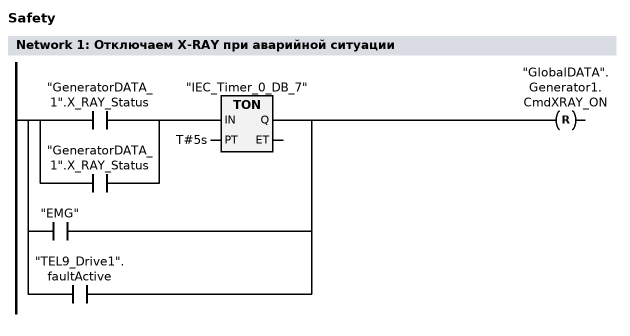
   "IEC_Timer_0_DB_7".TON(IN := "GeneratorDATA_1".X_RAY_Status OR "GeneratorDATA_1".X_RAY_Status, PT := T#5s);
   IF "IEC_Timer_0_DB_7".Q OR "EMG" OR "TEL9_Drive1".faultActive THEN
       "GlobalDATA".Generator1.CmdXRAY_ON := FALSE;
   END_IF;
END_REGION
END_FUNCTION_BLOCK

// folder: StatMachine

FUNCTION_BLOCK "StatMachineGLOBAL"   // FB6, SCL
{ S7_Optimized_Access := 'TRUE' }
VERSION : 0.1
   VAR
      Timer1 : Time;
      Timer2 : Time;
      PauseTime : Time := T#1000ms;
      preset_T_Prepare : Time := T#1m;
      preset_T_OpenDoor : Time := T#5s;
      T_Exposure : Time;
      T_Prepare : Time;
      sP1_Shutter1 : Bool;
      sP2_Shutter1 : Bool;
      sP1_Shutter2 : Bool;
      sP2_Shutter2 : Bool;
      sAbortPrepare : Bool;
      tempLAMP_XRAY : Bool;
      CareRay_Ready : Bool;
      door_opened : Bool;
      sForcePreset : Bool;
      sExposure : Bool;
      sScaning : Bool;
      sScaningOld : Bool;
      sShutter1_move : Bool;
      sShutter2_move : Bool;
      sScanComplite : Bool;
   END_VAR
BEGIN
   // Определяем сколько делается снимков
   IF "GlobalDATA".Generator1.Enable = TRUE AND "GlobalDATA".Generator2.Enable = TRUE THEN
       "GlobalDATA".CountShot := 2;
   ELSIF "GlobalDATA".Generator1.Enable = TRUE AND "GlobalDATA".Generator2.Enable = FALSE THEN
       "GlobalDATA".CountShot := 1;
   ELSIF "GlobalDATA".Generator1.Enable = FALSE AND "GlobalDATA".Generator2.Enable = TRUE THEN
       "GlobalDATA".CountShot := 1;
   ELSIF "GlobalDATA".Generator1.Enable = FALSE AND "GlobalDATA".Generator2.Enable = FALSE THEN
       "GlobalDATA".CountShot := 0;
   END_IF;

   // Формируем фронт сигнала для запуска импульсного таймера, формирующего импульс экспозиции (Trigger)
   IF #sScaningOld = #sScaning THEN
       #sScaning := FALSE;
   END_IF;

   // Если готовы привода шторок и генераторы то выставляем готовность
   IF ((("GlobalDATA".Generator1.Ready = TRUE AND "GlobalDATA".Shutter1.Ready AND "GlobalDATA".Generator1.Enable = TRUE)        //При активированом генераторе 1 должна быть готовность привода и генератора
       OR NOT "GlobalDATA".Generator1.Enable OR NOT "GlobalDATA".Scan_XRAY)                                                    //Если не используется генератор 1 или сканируем без X-RAY
       AND (("GlobalDATA".Generator2.Ready = TRUE AND "GlobalDATA".Shutter2.Ready AND "GlobalDATA".Generator2.Enable = TRUE)   //При активированом генераторе 2 должна быть готовность привода и генератора
       OR NOT "GlobalDATA".Generator2.Enable OR NOT "GlobalDATA".Scan_XRAY))                                                    //Если не используется генератор 2 или сканируем без X-RAY
       AND "GlobalDATA".CountShot > 0                                                                                           //Определено количество работающих генераторов
   THEN
       "GlobalDATA".readyToScan := TRUE;
   ELSE
       //Нет готовности к сканированию т.к. нет готовности одно из гнератора или привода шторки
       "GlobalDATA".readyToScan := FALSE;
   END_IF;

   //Режим работы сканера Ручной и Автоматический
   IF "GlobalDATA".modeScan="modeJOG"
       OR "GlobalDATA".modeScan="modeAUTO" THEN
       //Установка переменных, обязательных для режима JOG и AUTO
       "PresetAUTO_JOG"();

       //Обработка стадий cценария сканирования
       CASE "GlobalDATA".stageScan OF
           "stageWaitGuest":
               // Ожижание посетителя
               REGION Wait_Guest
                   "GlobalDATA".modeDrive := FALSE;
                   //Начало цикла сканирования когда шторка в первой позции для любого генератора
                   "GlobalDATA".Shutter1.cmdPOS1 := TRUE;
                   "GlobalDATA".Shutter1.cmdPOS2 := FALSE;
                   //Начало цикла сканирования когда шторка в первой позции для любого генератора
                   "GlobalDATA".Shutter2.cmdPOS1 := TRUE;
                   "GlobalDATA".Shutter2.cmdPOS2 := FALSE;
                   //Отключаем XRAY для всех генераторов
                   "GlobalDATA".Generator1.CmdXRAY_ON := FALSE;
                   "GlobalDATA".Generator2.CmdXRAY_ON := FALSE;

                   "GlobalDATA".newPreset := FALSE;    // Обнуляем признак получения нового пресета
                   "IR".SHOT_make := FALSE;            // Сбрасываем признак прихода нового посетителя
                   "K_Open_Door" := FALSE;             // Сбрасываем управление открытием двери

                   IF "IR".Guest_came                               // Пришел посетитель 
                       AND (("GlobalDATA".Shutter1.setPOS1 = TRUE  AND "GlobalDATA".Generator1.Enable = TRUE) OR "GlobalDATA".Generator1.Enable = FALSE)   // Шторка в исходной позиции если генератор 1 используется
                       AND (("GlobalDATA".Shutter2.setPOS1 = TRUE  AND "GlobalDATA".Generator2.Enable = TRUE) OR "GlobalDATA".Generator2.Enable = FALSE)   // Шторка в исходной позиции если генератор 2 используется
                       // OR внешнее событие для запуска сканирования. из UI команда на сканирование
                   THEN
                       IF "GlobalDATA".Scan_XRAY = TRUE                // Если сканируем с XRAY
                       THEN
                           //Устанавливаем пресет для первого генератора и включаем его
                           IF "GlobalDATA".Generator1.Enable = TRUE THEN
                               "LoadPresset"(N_Presset := "GlobalDATA".N_Presset,
                                             DATA_from := "PressetDATA".GUEST["GlobalDATA".N_Presset],
                                             DATA_to => "GeneratorDATA_1");
                               "GlobalDATA".Generator1.CmdXRAY_ON := TRUE;
                           END_IF;
                           //Устанавливаем пресет для второго генератора и включаем его
                           IF "GlobalDATA".Generator2.Enable = TRUE THEN
                               "LoadPresset"(N_Presset := "GlobalDATA".N_Presset,
                                             DATA_from := "PressetDATA".GUEST["GlobalDATA".N_Presset],
                                             DATA_to => "GeneratorDATA_2");
                               "GlobalDATA".Generator2.CmdXRAY_ON := TRUE;
                           END_IF;
                           #sAbortPrepare := FALSE;
                       ELSE
                           "GlobalDATA".stageScan := "stagePrepareScan";
                       END_IF;
                   END_IF;
               END_REGION Wait_Guest

           "stagePrepareScan":
               // Подготовка к сканированию
               REGION Prepare_Scan

                   "KM_Generator2" := #CareRay_Ready;
                   "GlobalDATA".readyData := FALSE;
                   #sScanComplite := FALSE; //Сброс признака готовности данных после выполнения снимка

                   IF #sAbortPrepare = TRUE THEN                               // Если принудительно прерван процесс сканирования. После срабатывания первого ИК датчика в течении 1 минуты нет никаких движений
                       #sAbortPrepare := FALSE;
                       "GlobalDATA".stageScan := "stageWaitGuest";
                       "IR".Guest_came := FALSE;
                       "GlobalDATA".Shutter1.cmdPOS1 := TRUE;
                       "GlobalDATA".Shutter1.cmdPOS2 := FALSE;
                       "GlobalDATA".Generator1.CmdXRAY_ON := FALSE;
                       "GlobalDATA".Shutter2.cmdPOS1 := TRUE;
                       "GlobalDATA".Shutter2.cmdPOS2 := FALSE;
                       "GlobalDATA".Generator2.CmdXRAY_ON := FALSE;
                   ELSIF ("IR".SHOT_make = TRUE OR "GlobalDATA".startScan)                                                                    // Если сработал второй инфракрасный датчик или принудительно запустили сканирование
                       AND ((#CareRay_Ready = TRUE AND ("GlobalDATA".newPreset = TRUE OR "GlobalDATA".startScan)) OR (#sForcePreset = TRUE))  // После распознания лица установили прессет в детекторе и панель CareRay готова
                       // Если получили новый пресет (распознали лицо)
                       // Если в течении установленного времени камера не распознала лицо
                       AND (("GlobalDATA".Generator1.XRAY_Status AND "GlobalDATA".Generator1.PWR_Status AND "GlobalDATA".Scan_XRAY AND "GlobalDATA".Generator1.Enable) OR NOT "GlobalDATA".Scan_XRAY OR NOT "GlobalDATA".Generator1.Enable)
                       AND (("GlobalDATA".Generator2.XRAY_Status AND "GlobalDATA".Generator2.PWR_Status AND "GlobalDATA".Scan_XRAY AND "GlobalDATA".Generator2.Enable) OR NOT "GlobalDATA".Scan_XRAY OR NOT "GlobalDATA".Generator2.Enable)
                       // Если генератор включен. X-RAY = TRUE
                       // Если фактическая мощность энергии генератора равна заанной
                       // Если сканируем с XRAY
                       // Или сканируем без XRAY и тогда не контролируем готовность генератора
                   THEN
                       //Перемещаем шторку первого генератора если генератор активен
                       IF "GlobalDATA".Generator1.Enable = TRUE THEN
                           "GlobalDATA".Shutter1.cmdPOS2 := TRUE;
                           "GlobalDATA".Shutter1.cmdPOS1 := FALSE;
                           #sShutter1_move := TRUE;
                           #sShutter2_move := FALSE;
                       //Перемещаем шторку второго генератора если генератор активен    
                       ELSIF "GlobalDATA".Generator2.Enable = TRUE THEN
                           "GlobalDATA".Shutter2.cmdPOS2 := FALSE;
                           "GlobalDATA".Shutter2.cmdPOS1 := FALSE;
                           #sShutter1_move := FALSE;
                           #sShutter2_move := TRUE;
                       END_IF;

                       //Устанавливаем время экспозиции
                       #T_Exposure := "PressetDATA".GUEST["GlobalDATA".N_Presset].Ttrigger;
                       "GlobalDATA".stageScan := "stageScaning";
                       #sScaning := TRUE;
                   END_IF;
               END_REGION Prepare_Scan

           "stageScaning":
               // Выполнение сканирования
               REGION Scaning

                   // Если первая шторка должна перемещаться, позиция достигнута, позиция установлена, завершена экспозиция (Trigger = OFF)
                   IF #sShutter1_move AND "TEL9_Drive1".targetPositionReached AND "GlobalDATA".Shutter1.setPOS2 AND #sExposure = FALSE
                   THEN
                       #sShutter1_move := FALSE;
                       "GlobalDATA".Generator1.CmdXRAY_ON := FALSE;
                       "GlobalDATA".Shutter1.cmdPOS2 := FALSE;
                       //Если активен второй генератор, то делаем второй снимок
                       IF "GlobalDATA".Generator2.Enable = TRUE THEN
                           "GlobalDATA".Shutter2.cmdPOS2 := TRUE;
                           "GlobalDATA".Shutter2.cmdPOS1 := FALSE;
                           #sShutter2_move := TRUE;
                           #sScaning := TRUE;
                       ELSE
                           "IR".Guest_came := FALSE;
                           "IR".SHOT_make := FALSE;
                           "GlobalDATA".Door.CmdOpen := TRUE;
                           "GlobalDATA".stageScan := "stageOpenDoor";
                           #door_opened := FALSE;
                           #sScaning := FALSE;
                           #sScanComplite := TRUE;     //Признак окончания сканирования
                           "GlobalDATA".startScan := FALSE;
                       END_IF;
                   END_IF;

                   // Если вторая шторка должна перемещаться, позиция достигнута, позиция установлена, завершена экспозиция (Trigger = OFF)
                   IF #sShutter2_move AND "TEL9_Drive2".targetPositionReached AND "GlobalDATA".Shutter2.setPOS2 AND #sExposure = FALSE
                   THEN
                       #sShutter2_move := FALSE;
                       "GlobalDATA".Generator2.CmdXRAY_ON := FALSE;
                       "GlobalDATA".Shutter2.cmdPOS2 := FALSE;
                       "IR".Guest_came := FALSE;
                       "IR".SHOT_make := FALSE;
                       "GlobalDATA".Door.CmdOpen := TRUE;
                       "GlobalDATA".stageScan := "stageOpenDoor";
                       #door_opened := FALSE;
                       #sScaning := FALSE;
                       #sScanComplite := TRUE;     //Признак окончания сканирования
                       "GlobalDATA".startScan := FALSE;
                   END_IF;
               END_REGION Scaning

           "stageOpenDoor":
               // Открытие двери
               REGION Open_Door    
                   IF ((#door_opened = TRUE AND "GlobalDATA".Door.CmdOpen = TRUE) OR (#door_opened = FALSE AND "GlobalDATA".Door.CmdOpen = FALSE)) // Если открылась дверь при наличии команды на открытие двери. Или дверь закрыта при отсутствии команды на открытие
                       AND (("GlobalDATA".Generator1.XRAY_Status = FALSE AND "GlobalDATA".Scan_XRAY = TRUE) OR ("GlobalDATA".Generator1.XRAY_Status = FALSE AND "GlobalDATA".Scan_XRAY = FALSE))
                   THEN
                       // Если открылась дверь
                       "K_Open_Door" := FALSE;
                       "GlobalDATA".Door.CmdOpen := FALSE;
                       "GlobalDATA".N_Presset := 1;
                       "GlobalDATA".Shutter1.cmdPOS1 := TRUE;
                       "GlobalDATA".Shutter1.cmdPOS2 := FALSE;
                   END_IF;

                   IF "GlobalDATA".Shutter1.setPOS1 = TRUE
                       AND "TEL9_Drive1".targetPositionReached = TRUE THEN
                       "GlobalDATA".Shutter1.cmdPOS1 := FALSE;
                       "IR".Guest_came := FALSE;
                       "IR".SHOT_make := FALSE;
                       "GlobalDATA".stageScan := "stageWaitGuest";
                   END_IF;
               END_REGION Open_Door   

           ELSE
               // Если не определен режим, то переходим в режим ожидания посетителя
               "GlobalDATA".stageScan := "stageWaitGuest";
       END_CASE;
   ELSE
       "IR".Guest_came := FALSE;
       "IR".SHOT_make := FALSE;
       "GlobalDATA".stageScan := "stageWaitGuest";
   END_IF;

   //Режим работы сканера Сервисный
   IF "GlobalDATA".modeScan = "modeSERVIСE" THEN
       //Установка переменных, обязательных для режима SERVICE
       "PresetSERVICE"();

       //Сервисный режим. Циклическое перемещение шторки 1
       REGION Cycle_Shutter 
           IF "GlobalDATA".Shutter1.cmdCycle THEN

               //Отключаем работу генератора
               "GlobalDATA".Generator1.CmdXRAY_ON := FALSE;
               //   проверяем отключен ли генератор
               IF "GeneratorDATA_1".X_RAY_Status = FALSE THEN
                   IF "GlobalDATA".Shutter1.setPOS1 = TRUE AND "TEL9_Drive1".targetPositionReached = TRUE THEN
                       #sP2_Shutter1 := TRUE;
                       #sP1_Shutter1 := FALSE;
                   ELSIF "GlobalDATA".Shutter1.setPOS2 = TRUE AND "TEL9_Drive1".targetPositionReached = TRUE THEN
                       #sP1_Shutter1 := TRUE;
                       #sP2_Shutter1 := FALSE;
                   END_IF;
                   //Пауза в крайней точке при циклическом перемещении шторки 1
                   "IEC_Timer_0_DB_2".TON(IN := #sP2_Shutter1,
                                          PT := #PauseTime,
                                          Q => "GlobalDATA".Shutter1.cmdPOS2,
                                          ET => #Timer1);

                   "IEC_Timer_0_DB_4".TON(IN := #sP1_Shutter1,
                                          PT := #PauseTime,
                                          Q => "GlobalDATA".Shutter1.cmdPOS1,
                                          ET => #Timer2);
               END_IF;
           END_IF;
           //Сервисный режим. Циклическое перемещение шторки 1
           IF "GlobalDATA".Shutter2.cmdCycle THEN
               //Отключаем работу генератора
               "GlobalDATA".Generator2.CmdXRAY_ON := FALSE;
               //   проверяем отключен ли генератор
               IF "GeneratorDATA_2".X_RAY_Status = FALSE THEN
                   IF "GlobalDATA".Shutter2.setPOS1 = TRUE AND "TEL9_Drive2".targetPositionReached = TRUE THEN
                       #sP2_Shutter2 := TRUE;
                       #sP1_Shutter2 := FALSE;
                   ELSIF "GlobalDATA".Shutter2.setPOS2 = TRUE AND "TEL9_Drive2".targetPositionReached = TRUE THEN
                       #sP1_Shutter2 := TRUE;
                       #sP2_Shutter2 := FALSE;
                   END_IF;
                   //Пауза в крайней точке при циклическом перемещении шторки 2
                   "IEC_Timer_0_DB_13".TON(IN:=#sP2_Shutter2,
                                           PT:=#PauseTime,
                                           Q=>"GlobalDATA".Shutter2.cmdPOS2);

                   "IEC_Timer_0_DB_14".TON(IN := #sP1_Shutter2,
                                           PT := #PauseTime,
                                           Q => "GlobalDATA".Shutter2.cmdPOS1);
               END_IF;
           END_IF;
       END_REGION Cycle_Shutter

   END_IF;

   // Режим ограниченных возможностей сканера
   IF "GlobalDATA".modeScan = "modeLIMITED" THEN
       "GlobalDATA".readyData := FALSE;
       "GlobalDATA".stageScan := "stageWaitGuest";
       "GlobalDATA".newPreset := FALSE;
   END_IF;

   // Режим отключенного сканера
   IF "GlobalDATA".modeScan="modeOFF" THEN
       //Установки для режима отключено
       "PresetOFF"();
       "GlobalDATA".stageScan := "stageWaitGuest";
   END_IF;

   // Таймер отсчета времени открытия двери. Косвенный контроль. Просто выдерживаем время после подачи команды на открытие двери, считая при этом, что дверь открыта
   "IEC_Timer_0_DB_5".TON(IN := "GlobalDATA".Door.CmdOpen,
                          PT := #preset_T_OpenDoor,
                          Q => #door_opened);

   // Симуляция готовности панели детекторов. По итогу должны контролировать дискретный сигнал от Control Box (Ready)
   "IEC_Timer_0_DB_8".TON(IN := "GlobalDATA".newPreset,
                          PT := T#2s,
                          Q => #CareRay_Ready);

   // Таймер контроля прихода посетителя. Если сработал только первый ИК датчик и нет никаких движений то по таймеру сбрасываем цикл на исходную позицию
   "IEC_Timer_0_DB_6".TON(IN:="IR".Guest_came,
                      PT:=T#10m,
                      Q=>#sAbortPrepare);

   // После прихода посетителя если он не идентифицирован для установки прессета, то через интервальный таймер принудительно устанавливаем прессет
   "IEC_Timer_0_DB_11".TON(IN:="IR".Guest_came,
                           PT:=T#5s,
                           Q=>#sForcePreset);

   // Импульс Trigger для экспозиции. Запуск по фронту
   "IEC_Timer_0_DB_15".TP(IN:=#sScaning,
                          PT:=#T_Exposure,
                          Q=>#sExposure);
   #sScaningOld := #sScaning;

   // Имитация сигнала Ready по готовности данных CaryRay
   "IEC_Timer_0_DB_16".TON(IN := #sScanComplite,
                           PT := T#500ms,
                           Q=> "GlobalDATA".readyData);


   // Обновляем выходные переменные
   "KM_Generator2" := #CareRay_Ready;
   "K_Open_Door" := "GlobalDATA".Door.CmdOpen;
   "TRIG_Detectors" := #sExposure;                 //Устанавливаем сигнал Trigger для CareRay
END_FUNCTION_BLOCK

FUNCTION "PresetAUTO_JOG" : Void   // FC13, SCL
{ S7_Optimized_Access := 'TRUE' }
VERSION : 0.1
BEGIN
       //Включаем разрешение работы привода
       "GlobalDATA".Shutter1.cmdOFF1 := TRUE;
       "GlobalDATA".Shutter2.cmdOFF1 := TRUE;

       //Блокируем циклическое перемещение шторки
       "GlobalDATA".Shutter1.cmdCycle := FALSE;
       "GlobalDATA".Shutter2.cmdCycle := FALSE;
       "GlobalDATA".modeDrive := FALSE;
END_FUNCTION

FUNCTION "PresetSERVICE" : Void   // FC14, SCL
{ S7_Optimized_Access := 'TRUE' }
VERSION : 0.1
BEGIN
   //Устанавливаем разрешения работы приводов
   "GlobalDATA".Shutter1.cmdOFF1 := TRUE;
   "GlobalDATA".Shutter2.cmdOFF1 := TRUE;
END_FUNCTION

FUNCTION "PresetOFF" : Void   // FC15, SCL
{ S7_Optimized_Access := 'TRUE' }
VERSION : 0.1
BEGIN
   //Устанавливаем разрешения работы привода 1
   "GlobalDATA".Shutter1.cmdOFF1 := FALSE;
   "GlobalDATA".Shutter1.cmdCycle := FALSE;
   "GlobalDATA".Shutter1.cmdPOS1 := FALSE;
   "GlobalDATA".Shutter1.cmdPOS2 := FALSE;

   //Устанавливаем разрешения работы привода 2
   "GlobalDATA".Shutter2.cmdOFF1 := FALSE;
   "GlobalDATA".Shutter2.cmdCycle := FALSE;
   "GlobalDATA".Shutter2.cmdPOS1 := FALSE;
   "GlobalDATA".Shutter2.cmdPOS2 := FALSE;

   //Устанавливаем режим работы для генератора 1
   "GlobalDATA".Generator1.CmdXRAY_ON := FALSE;
   "GlobalDATA".Generator1.cmdWarm := 0;

   //Устанавливаем режим работы для генератора 2
   "GlobalDATA".Generator2.CmdXRAY_ON := FALSE;
   "GlobalDATA".Generator2.cmdWarm := 0;

   "GlobalDATA".stageScan := "stageWaitGuest";
   "GlobalDATA".newPreset := FALSE;
END_FUNCTION